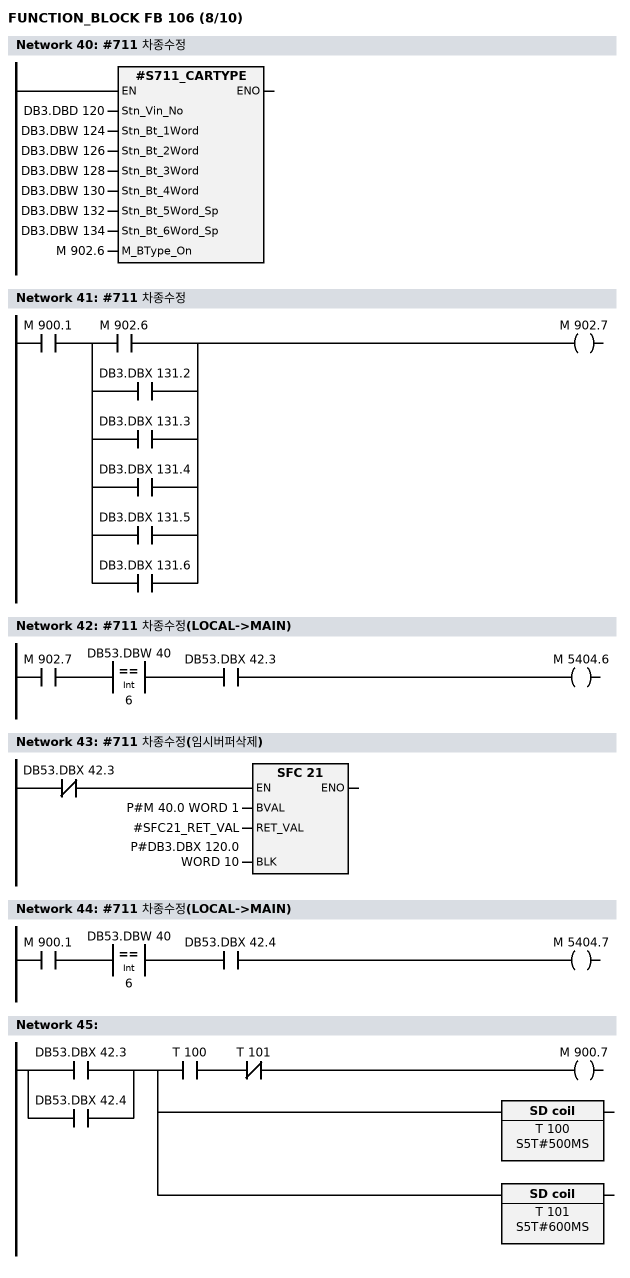

      CALL #S711_CARTYPE (
           Stn_Vin_No               := DB3.DBD  120,
           Stn_Bt_1Word             := DB3.DBW  124,
           Stn_Bt_2Word             := DB3.DBW  126,
           Stn_Bt_3Word             := DB3.DBW  128,
           Stn_Bt_4Word             := DB3.DBW  130,
           Stn_Bt_5Word_Sp          := DB3.DBW  132,
           Stn_Bt_6Word_Sp          := DB3.DBW  134,
           M_BType_On               := M    902.6);

      NOP   0;
NETWORK
TITLE =#711 차종수정

      A     M    900.1;
      A(    ;
      O     M    902.6;
      O     DB3.DBX  131.2;
      O     DB3.DBX  131.3;
      O     DB3.DBX  131.4;
      O     DB3.DBX  131.5;
      O     DB3.DBX  131.6;
      )     ;
      =     M    902.7;
NETWORK
TITLE =#711 차종수정(LOCAL->MAIN)

      A     M    902.7;
      A(    ;
      L     DB53.DBW   40;
      L     6;
      ==I   ;
      )     ;
      A     DB53.DBX   42.3;
      =     M   5404.6;
NETWORK
TITLE =#711 차종수정(임시버퍼삭제)

      AN    DB53.DBX   42.3;
      JNB   _00c;
      CALL SFC   21 (
           BVAL                     := P#M 40.0 WORD 1,
           RET_VAL                  := #SFC21_RET_VAL,
           BLK                      := P#DB3.DBX 120.0 WORD 10);
_00c: NOP   0;
NETWORK
TITLE =#711 차종수정(LOCAL->MAIN)

      A     M    900.1;
      A(    ;
      L     DB53.DBW   40;
      L     6;
      ==I   ;
      )     ;
      A     DB53.DBX   42.4;
      =     M   5404.7;
NETWORK
TITLE =

      O     DB53.DBX   42.3;
      O     DB53.DBX   42.4;
      =     L      2.0;
      A     L      2.0;
      A     T    100;
      AN    T    101;
      =     M    900.7;
      A     L      2.0;
      BLD   102;
      L     S5T#500MS;
      SD    T    100;
      A     L      2.0;
      BLD   102;
      L     S5T#600MS;
      SD    T    101;
NETWORK
TITLE =
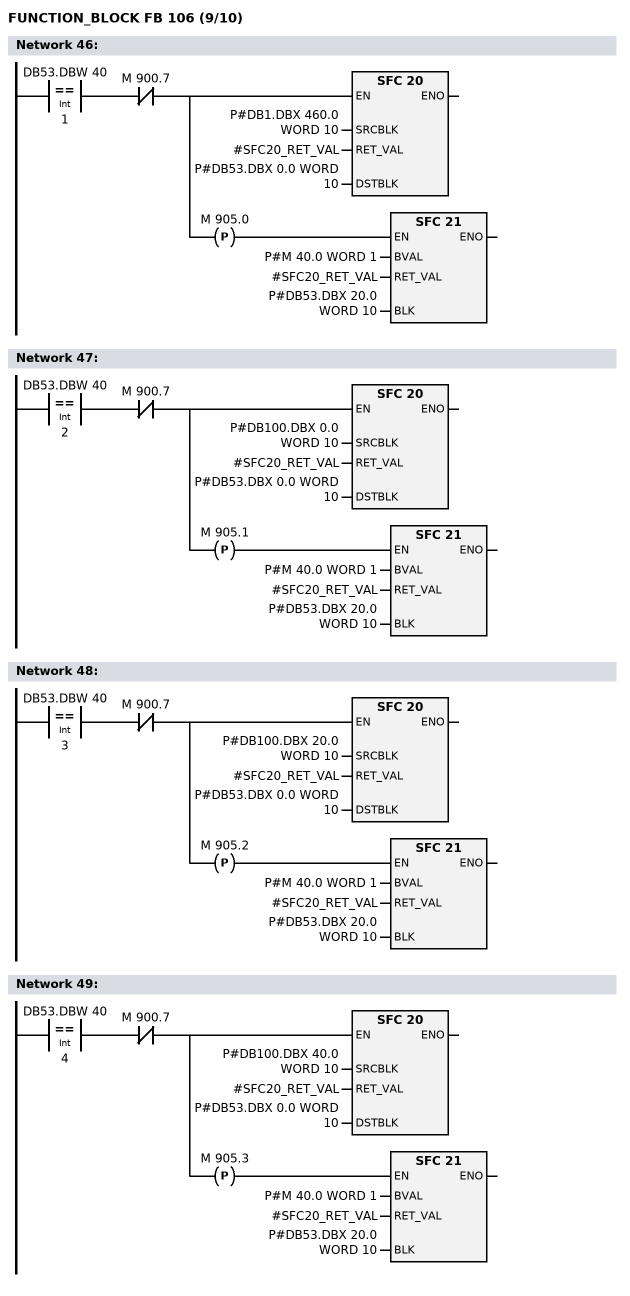

      A(    ;
      L     DB53.DBW   40;
      L     1;
      ==I   ;
      )     ;
      AN    M    900.7;
      =     L      2.0;
      A     L      2.0;
      JNB   _00d;
      CALL SFC   20 (
           SRCBLK                   := P#DB1.DBX 460.0 WORD 10,
           RET_VAL                  := #SFC20_RET_VAL,
           DSTBLK                   := P#DB53.DBX 0.0 WORD 10);
_00d: NOP   0;
      A     L      2.0;
      FP    M    905.0;
      JNB   _00e;
      CALL SFC   21 (
           BVAL                     := P#M 40.0 WORD 1,
           RET_VAL                  := #SFC20_RET_VAL,
           BLK                      := P#DB53.DBX 20.0 WORD 10);
_00e: NOP   0;
NETWORK
TITLE =

      A(    ;
      L     DB53.DBW   40;
      L     2;
      ==I   ;
      )     ;
      AN    M    900.7;
      =     L      2.0;
      A     L      2.0;
      JNB   _00f;
      CALL SFC   20 (
           SRCBLK                   := P#DB100.DBX 0.0 WORD 10,
           RET_VAL                  := #SFC20_RET_VAL,
           DSTBLK                   := P#DB53.DBX 0.0 WORD 10);
_00f: NOP   0;
      A     L      2.0;
      FP    M    905.1;
      JNB   _010;
      CALL SFC   21 (
           BVAL                     := P#M 40.0 WORD 1,
           RET_VAL                  := #SFC20_RET_VAL,
           BLK                      := P#DB53.DBX 20.0 WORD 10);
_010: NOP   0;
NETWORK
TITLE =

      A(    ;
      L     DB53.DBW   40;
      L     3;
      ==I   ;
      )     ;
      AN    M    900.7;
      =     L      2.0;
      A     L      2.0;
      JNB   _011;
      CALL SFC   20 (
           SRCBLK                   := P#DB100.DBX 20.0 WORD 10,
           RET_VAL                  := #SFC20_RET_VAL,
           DSTBLK                   := P#DB53.DBX 0.0 WORD 10);
_011: NOP   0;
      A     L      2.0;
      FP    M    905.2;
      JNB   _012;
      CALL SFC   21 (
           BVAL                     := P#M 40.0 WORD 1,
           RET_VAL                  := #SFC20_RET_VAL,
           BLK                      := P#DB53.DBX 20.0 WORD 10);
_012: NOP   0;
NETWORK
TITLE =

      A(    ;
      L     DB53.DBW   40;
      L     4;
      ==I   ;
      )     ;
      AN    M    900.7;
      =     L      2.0;
      A     L      2.0;
      JNB   _013;
      CALL SFC   20 (
           SRCBLK                   := P#DB100.DBX 40.0 WORD 10,
           RET_VAL                  := #SFC20_RET_VAL,
           DSTBLK                   := P#DB53.DBX 0.0 WORD 10);
_013: NOP   0;
      A     L      2.0;
      FP    M    905.3;
      JNB   _014;
      CALL SFC   21 (
           BVAL                     := P#M 40.0 WORD 1,
           RET_VAL                  := #SFC20_RET_VAL,
           BLK                      := P#DB53.DBX 20.0 WORD 10);
_014: NOP   0;
NETWORK
TITLE =
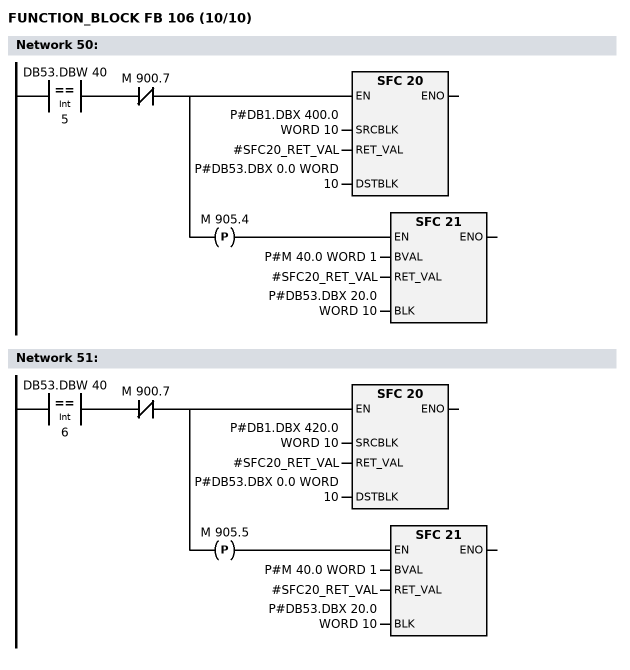

      A(    ;
      L     DB53.DBW   40;
      L     5;
      ==I   ;
      )     ;
      AN    M    900.7;
      =     L      2.0;
      A     L      2.0;
      JNB   _015;
      CALL SFC   20 (
           SRCBLK                   := P#DB1.DBX 400.0 WORD 10,
           RET_VAL                  := #SFC20_RET_VAL,
           DSTBLK                   := P#DB53.DBX 0.0 WORD 10);
_015: NOP   0;
      A     L      2.0;
      FP    M    905.4;
      JNB   _016;
      CALL SFC   21 (
           BVAL                     := P#M 40.0 WORD 1,
           RET_VAL                  := #SFC20_RET_VAL,
           BLK                      := P#DB53.DBX 20.0 WORD 10);
_016: NOP   0;
NETWORK
TITLE =

      A(    ;
      L     DB53.DBW   40;
      L     6;
      ==I   ;
      )     ;
      AN    M    900.7;
      =     L      2.0;
      A     L      2.0;
      JNB   _017;
      CALL SFC   20 (
           SRCBLK                   := P#DB1.DBX 420.0 WORD 10,
           RET_VAL                  := #SFC20_RET_VAL,
           DSTBLK                   := P#DB53.DBX 0.0 WORD 10);
_017: NOP   0;
      A     L      2.0;
      FP    M    905.5;
      JNB   _018;
      CALL SFC   21 (
           BVAL                     := P#M 40.0 WORD 1,
           RET_VAL                  := #SFC20_RET_VAL,
           BLK                      := P#DB53.DBX 20.0 WORD 10);
_018: NOP   0;
END_FUNCTION_BLOCK

DATA_BLOCK DB 106
TITLE =
VERSION : 0.0

 FB 106
BEGIN
   CAR_TYPE_MODIFY.Station := 0;
   CAR_TYPE_MODIFY.HMI_Disp_DB := 0;
   CAR_TYPE_MODIFY.HMI_Disp_Add := 0;
   CAR_TYPE_MODIFY.CType_DB := 0;
   CAR_TYPE_MODIFY.CType_Start_Add := 0;
   CAR_TYPE_MODIFY.Byte_per_Stn := 0;
   CAR_TYPE_MODIFY.M_Modify_OK := FALSE;
   CAR_TYPE_MODIFY.SS_CCR_On := FALSE;
   CAR_TYPE_MODIFY.PB_Set := FALSE;
   CAR_TYPE_MODIFY.PB_Reset := FALSE;
   CAR_TYPE_MODIFY.LP_CCR_On := FALSE;
   CAR_TYPE_MODIFY.LP_Modify_On := FALSE;
   CAR_TYPE_MODIFY.Source_Data := W#16#0;
   CAR_TYPE_MODIFY.Modify_Data := W#16#0;
   CAR_TYPE_MODIFY.Pre_Station := 0;
   CAR_TYPE_MODIFY.Station_PLS := FALSE;
   CAR_TYPE_MODIFY.Source_Add := 0;
   CAR_TYPE_MODIFY.SFC20_Ret := 0;
   CAR_TYPE_MODIFY.Fill_Source := W#16#0;
   SFC20_RET_VAL := 0;
   HMI_CAR_TYPE_V2.Stn_Vin_No := L#0;
   HMI_CAR_TYPE_V2.Stn_Bt_1Word := W#16#0;
   HMI_CAR_TYPE_V2.Stn_Bt_2Word := W#16#0;
   HMI_CAR_TYPE_V2.Stn_Bt_3Word := W#16#0;
   HMI_CAR_TYPE_V2.Stn_Bt_4Word := W#16#0;
   HMI_CAR_TYPE_V2.Stn_Bt_5Word_Sp := W#16#0;
   HMI_CAR_TYPE_V2.Stn_Bt_6Word_Sp := W#16#0;
   HMI_CAR_TYPE_V2.M_BType_On := FALSE;
   HMI_CAR_TYPE_V2.M_BType_None := FALSE;
   HMI_CAR_TYPE_V2.M_Bypass_BType := FALSE;
   HMI_CAR_TYPE_V2.M_BType_TL := FALSE;
   HMI_CAR_TYPE_V2.M_BType_LM := FALSE;
   HMI_CAR_TYPE_V2.M_BType_SP1 := FALSE;
   HMI_CAR_TYPE_V2.M_BType_SP2 := FALSE;
   HMI_CAR_TYPE_V2.M_BType_SP3 := FALSE;
   HMI_CAR_TYPE_V2.M_BType_DOM := FALSE;
   HMI_CAR_TYPE_V2.M_BType_EXP := FALSE;
   HMI_CAR_TYPE_V2.Robot_Prog_No := 0;
   HMI_CAR_TYPE_V2.STN_Btype_1Arr[0] := FALSE;
   HMI_CAR_TYPE_V2.STN_Btype_1Arr[1] := FALSE;
   HMI_CAR_TYPE_V2.STN_Btype_1Arr[2] := FALSE;
   HMI_CAR_TYPE_V2.STN_Btype_1Arr[3] := FALSE;
   HMI_CAR_TYPE_V2.STN_Btype_1Arr[4] := FALSE;
   HMI_CAR_TYPE_V2.STN_Btype_1Arr[5] := FALSE;
   HMI_CAR_TYPE_V2.STN_Btype_1Arr[6] := FALSE;
   HMI_CAR_TYPE_V2.STN_Btype_1Arr[7] := FALSE;
   HMI_CAR_TYPE_V2.STN_Btype_1Arr[8] := FALSE;
   HMI_CAR_TYPE_V2.STN_Btype_1Arr[9] := FALSE;
   HMI_CAR_TYPE_V2.STN_Btype_1Arr[10] := FALSE;
   HMI_CAR_TYPE_V2.STN_Btype_1Arr[11] := FALSE;
   HMI_CAR_TYPE_V2.STN_Btype_1Arr[12] := FALSE;
   HMI_CAR_TYPE_V2.STN_Btype_1Arr[13] := FALSE;
   HMI_CAR_TYPE_V2.STN_Btype_1Arr[14] := FALSE;
   HMI_CAR_TYPE_V2.STN_Btype_1Arr[15] := FALSE;
   HMI_CAR_TYPE_V2.STN_Btype_2Arr[0] := FALSE;
   HMI_CAR_TYPE_V2.STN_Btype_2Arr[1] := FALSE;
   HMI_CAR_TYPE_V2.STN_Btype_2Arr[2] := FALSE;
   HMI_CAR_TYPE_V2.STN_Btype_2Arr[3] := FALSE;
   HMI_CAR_TYPE_V2.STN_Btype_2Arr[4] := FALSE;
   HMI_CAR_TYPE_V2.STN_Btype_2Arr[5] := FALSE;
   HMI_CAR_TYPE_V2.STN_Btype_2Arr[6] := FALSE;
   HMI_CAR_TYPE_V2.STN_Btype_2Arr[7] := FALSE;
   HMI_CAR_TYPE_V2.STN_Btype_2Arr[8] := FALSE;
   HMI_CAR_TYPE_V2.STN_Btype_2Arr[9] := FALSE;
   HMI_CAR_TYPE_V2.STN_Btype_2Arr[10] := FALSE;
   HMI_CAR_TYPE_V2.STN_Btype_2Arr[11] := FALSE;
   HMI_CAR_TYPE_V2.STN_Btype_2Arr[12] := FALSE;
   HMI_CAR_TYPE_V2.STN_Btype_2Arr[13] := FALSE;
   HMI_CAR_TYPE_V2.STN_Btype_2Arr[14] := FALSE;
   HMI_CAR_TYPE_V2.STN_Btype_2Arr[15] := FALSE;
   HMI_CAR_TYPE_V2.STN_Btype_3Arr[0] := FALSE;
   HMI_CAR_TYPE_V2.STN_Btype_3Arr[1] := FALSE;
   HMI_CAR_TYPE_V2.STN_Btype_3Arr[2] := FALSE;
   HMI_CAR_TYPE_V2.STN_Btype_3Arr[3] := FALSE;
   HMI_CAR_TYPE_V2.STN_Btype_3Arr[4] := FALSE;
   HMI_CAR_TYPE_V2.STN_Btype_3Arr[5] := FALSE;
   HMI_CAR_TYPE_V2.STN_Btype_3Arr[6] := FALSE;
   HMI_CAR_TYPE_V2.STN_Btype_3Arr[7] := FALSE;
   HMI_CAR_TYPE_V2.STN_Btype_3Arr[8] := FALSE;
   HMI_CAR_TYPE_V2.STN_Btype_3Arr[9] := FALSE;
   HMI_CAR_TYPE_V2.STN_Btype_3Arr[10] := FALSE;
   HMI_CAR_TYPE_V2.STN_Btype_3Arr[11] := FALSE;
   HMI_CAR_TYPE_V2.STN_Btype_3Arr[12] := FALSE;
   HMI_CAR_TYPE_V2.STN_Btype_3Arr[13] := FALSE;
   HMI_CAR_TYPE_V2.STN_Btype_3Arr[14] := FALSE;
   HMI_CAR_TYPE_V2.STN_Btype_3Arr[15] := FALSE;
   HMI_CAR_TYPE_V2.STN_Btype_4Arr[0] := FALSE;
   HMI_CAR_TYPE_V2.STN_Btype_4Arr[1] := FALSE;
   HMI_CAR_TYPE_V2.STN_Btype_4Arr[2] := FALSE;
   HMI_CAR_TYPE_V2.STN_Btype_4Arr[3] := FALSE;
   HMI_CAR_TYPE_V2.STN_Btype_4Arr[4] := FALSE;
   HMI_CAR_TYPE_V2.STN_Btype_4Arr[5] := FALSE;
   HMI_CAR_TYPE_V2.STN_Btype_4Arr[6] := FALSE;
   HMI_CAR_TYPE_V2.STN_Btype_4Arr[7] := FALSE;
   HMI_CAR_TYPE_V2.STN_Btype_4Arr[8] := FALSE;
   HMI_CAR_TYPE_V2.STN_Btype_4Arr[9] := FALSE;
   HMI_CAR_TYPE_V2.STN_Btype_4Arr[10] := FALSE;
   HMI_CAR_TYPE_V2.STN_Btype_4Arr[11] := FALSE;
   HMI_CAR_TYPE_V2.STN_Btype_4Arr[12] := FALSE;
   HMI_CAR_TYPE_V2.STN_Btype_4Arr[13] := FALSE;
   HMI_CAR_TYPE_V2.STN_Btype_4Arr[14] := FALSE;
   HMI_CAR_TYPE_V2.STN_Btype_4Arr[15] := FALSE;
   HMI_CAR_TYPE_V2.STN_Btype_5Arr[0] := FALSE;
   HMI_CAR_TYPE_V2.STN_Btype_5Arr[1] := FALSE;
   HMI_CAR_TYPE_V2.STN_Btype_5Arr[2] := FALSE;
   HMI_CAR_TYPE_V2.STN_Btype_5Arr[3] := FALSE;
   HMI_CAR_TYPE_V2.STN_Btype_5Arr[4] := FALSE;
   HMI_CAR_TYPE_V2.STN_Btype_5Arr[5] := FALSE;
   HMI_CAR_TYPE_V2.STN_Btype_5Arr[6] := FALSE;
   HMI_CAR_TYPE_V2.STN_Btype_5Arr[7] := FALSE;
   HMI_CAR_TYPE_V2.STN_Btype_5Arr[8] := FALSE;
   HMI_CAR_TYPE_V2.STN_Btype_5Arr[9] := FALSE;
   HMI_CAR_TYPE_V2.STN_Btype_5Arr[10] := FALSE;
   HMI_CAR_TYPE_V2.STN_Btype_5Arr[11] := FALSE;
   HMI_CAR_TYPE_V2.STN_Btype_5Arr[12] := FALSE;
   HMI_CAR_TYPE_V2.STN_Btype_5Arr[13] := FALSE;
   HMI_CAR_TYPE_V2.STN_Btype_5Arr[14] := FALSE;
   HMI_CAR_TYPE_V2.STN_Btype_5Arr[15] := FALSE;
   HMI_CAR_TYPE_V2.STN_Btype_6Arr[0] := FALSE;
   HMI_CAR_TYPE_V2.STN_Btype_6Arr[1] := FALSE;
   HMI_CAR_TYPE_V2.STN_Btype_6Arr[2] := FALSE;
   HMI_CAR_TYPE_V2.STN_Btype_6Arr[3] := FALSE;
   HMI_CAR_TYPE_V2.STN_Btype_6Arr[4] := FALSE;
   HMI_CAR_TYPE_V2.STN_Btype_6Arr[5] := FALSE;
   HMI_CAR_TYPE_V2.STN_Btype_6Arr[6] := FALSE;
   HMI_CAR_TYPE_V2.STN_Btype_6Arr[7] := FALSE;
   HMI_CAR_TYPE_V2.STN_Btype_6Arr[8] := FALSE;
   HMI_CAR_TYPE_V2.STN_Btype_6Arr[9] := FALSE;
   HMI_CAR_TYPE_V2.STN_Btype_6Arr[10] := FALSE;
   HMI_CAR_TYPE_V2.STN_Btype_6Arr[11] := FALSE;
   HMI_CAR_TYPE_V2.STN_Btype_6Arr[12] := FALSE;
   HMI_CAR_TYPE_V2.STN_Btype_6Arr[13] := FALSE;
   HMI_CAR_TYPE_V2.STN_Btype_6Arr[14] := FALSE;
   HMI_CAR_TYPE_V2.STN_Btype_6Arr[15] := FALSE;
   HMI_CAR_TYPE_V2.STN_1st_BT_On := FALSE;
   HMI_CAR_TYPE_V2.STN_2nd_BT_On := FALSE;
   HMI_CAR_TYPE_V2.STN_3rd_BT_On := FALSE;
   HMI_CAR_TYPE_V2.STN_4th_BT_On := FALSE;
   HMI_CAR_TYPE_V2.STN_5th_BT_On := FALSE;
   HMI_CAR_TYPE_V2.STN_6th_BT_On := FALSE;
   HMI_CAR_TYPE_V2.STN_7th_BT_On := FALSE;
   HMI_CAR_TYPE_V2.STN_8th_BT_On := FALSE;
   HMI_CAR_TYPE_V2.STN_9th_BT_On := FALSE;
   HMI_CAR_TYPE_V2.STN_10th_BT_On := FALSE;
   HMI_CAR_TYPE_V2.STN_11th_BT_On := FALSE;
   HMI_CAR_TYPE_V2.STN_12th_BT_On := FALSE;
   HMI_CAR_TYPE_V2.STN_1st_BT_Off := FALSE;
   HMI_CAR_TYPE_V2.BLKMove_Ret := 0;
   HMI_CAR_TYPE_V2.VIN_1BCD := W#16#0;
   HMI_CAR_TYPE_V2.VIN_2BCD := W#16#0;
   HMI_CAR_TYPE_V2.VIN_1Int := 0;
   HMI_CAR_TYPE_V2.VIN_2Int := 0;
   S6_HMI_CAR_TYPE_V2.Stn_Vin_No := L#0;
   S6_HMI_CAR_TYPE_V2.Stn_Bt_1Word := W#16#0;
   S6_HMI_CAR_TYPE_V2.Stn_Bt_2Word := W#16#0;
   S6_HMI_CAR_TYPE_V2.Stn_Bt_3Word := W#16#0;
   S6_HMI_CAR_TYPE_V2.Stn_Bt_4Word := W#16#0;
   S6_HMI_CAR_TYPE_V2.Stn_Bt_5Word_Sp := W#16#0;
   S6_HMI_CAR_TYPE_V2.Stn_Bt_6Word_Sp := W#16#0;
   S6_HMI_CAR_TYPE_V2.M_BType_On := FALSE;
   S6_HMI_CAR_TYPE_V2.M_BType_None := FALSE;
   S6_HMI_CAR_TYPE_V2.M_Bypass_BType := FALSE;
   S6_HMI_CAR_TYPE_V2.M_BType_TL := FALSE;
   S6_HMI_CAR_TYPE_V2.M_BType_LM := FALSE;
   S6_HMI_CAR_TYPE_V2.M_BType_SP1 := FALSE;
   S6_HMI_CAR_TYPE_V2.M_BType_SP2 := FALSE;
   S6_HMI_CAR_TYPE_V2.M_BType_SP3 := FALSE;
   S6_HMI_CAR_TYPE_V2.M_BType_DOM := FALSE;
   S6_HMI_CAR_TYPE_V2.M_BType_EXP := FALSE;
   S6_HMI_CAR_TYPE_V2.Robot_Prog_No := 0;
   S6_HMI_CAR_TYPE_V2.STN_Btype_1Arr[0] := FALSE;
   S6_HMI_CAR_TYPE_V2.STN_Btype_1Arr[1] := FALSE;
   S6_HMI_CAR_TYPE_V2.STN_Btype_1Arr[2] := FALSE;
   S6_HMI_CAR_TYPE_V2.STN_Btype_1Arr[3] := FALSE;
   S6_HMI_CAR_TYPE_V2.STN_Btype_1Arr[4] := FALSE;
   S6_HMI_CAR_TYPE_V2.STN_Btype_1Arr[5] := FALSE;
   S6_HMI_CAR_TYPE_V2.STN_Btype_1Arr[6] := FALSE;
   S6_HMI_CAR_TYPE_V2.STN_Btype_1Arr[7] := FALSE;
   S6_HMI_CAR_TYPE_V2.STN_Btype_1Arr[8] := FALSE;
   S6_HMI_CAR_TYPE_V2.STN_Btype_1Arr[9] := FALSE;
   S6_HMI_CAR_TYPE_V2.STN_Btype_1Arr[10] := FALSE;
   S6_HMI_CAR_TYPE_V2.STN_Btype_1Arr[11] := FALSE;
   S6_HMI_CAR_TYPE_V2.STN_Btype_1Arr[12] := FALSE;
   S6_HMI_CAR_TYPE_V2.STN_Btype_1Arr[13] := FALSE;
   S6_HMI_CAR_TYPE_V2.STN_Btype_1Arr[14] := FALSE;
   S6_HMI_CAR_TYPE_V2.STN_Btype_1Arr[15] := FALSE;
   S6_HMI_CAR_TYPE_V2.STN_Btype_2Arr[0] := FALSE;
   S6_HMI_CAR_TYPE_V2.STN_Btype_2Arr[1] := FALSE;
   S6_HMI_CAR_TYPE_V2.STN_Btype_2Arr[2] := FALSE;
   S6_HMI_CAR_TYPE_V2.STN_Btype_2Arr[3] := FALSE;
   S6_HMI_CAR_TYPE_V2.STN_Btype_2Arr[4] := FALSE;
   S6_HMI_CAR_TYPE_V2.STN_Btype_2Arr[5] := FALSE;
   S6_HMI_CAR_TYPE_V2.STN_Btype_2Arr[6] := FALSE;
   S6_HMI_CAR_TYPE_V2.STN_Btype_2Arr[7] := FALSE;
   S6_HMI_CAR_TYPE_V2.STN_Btype_2Arr[8] := FALSE;
   S6_HMI_CAR_TYPE_V2.STN_Btype_2Arr[9] := FALSE;
   S6_HMI_CAR_TYPE_V2.STN_Btype_2Arr[10] := FALSE;
   S6_HMI_CAR_TYPE_V2.STN_Btype_2Arr[11] := FALSE;
   S6_HMI_CAR_TYPE_V2.STN_Btype_2Arr[12] := FALSE;
   S6_HMI_CAR_TYPE_V2.STN_Btype_2Arr[13] := FALSE;
   S6_HMI_CAR_TYPE_V2.STN_Btype_2Arr[14] := FALSE;
   S6_HMI_CAR_TYPE_V2.STN_Btype_2Arr[15] := FALSE;
   S6_HMI_CAR_TYPE_V2.STN_Btype_3Arr[0] := FALSE;
   S6_HMI_CAR_TYPE_V2.STN_Btype_3Arr[1] := FALSE;
   S6_HMI_CAR_TYPE_V2.STN_Btype_3Arr[2] := FALSE;
   S6_HMI_CAR_TYPE_V2.STN_Btype_3Arr[3] := FALSE;
   S6_HMI_CAR_TYPE_V2.STN_Btype_3Arr[4] := FALSE;
   S6_HMI_CAR_TYPE_V2.STN_Btype_3Arr[5] := FALSE;
   S6_HMI_CAR_TYPE_V2.STN_Btype_3Arr[6] := FALSE;
   S6_HMI_CAR_TYPE_V2.STN_Btype_3Arr[7] := FALSE;
   S6_HMI_CAR_TYPE_V2.STN_Btype_3Arr[8] := FALSE;
   S6_HMI_CAR_TYPE_V2.STN_Btype_3Arr[9] := FALSE;
   S6_HMI_CAR_TYPE_V2.STN_Btype_3Arr[10] := FALSE;
   S6_HMI_CAR_TYPE_V2.STN_Btype_3Arr[11] := FALSE;
   S6_HMI_CAR_TYPE_V2.STN_Btype_3Arr[12] := FALSE;
   S6_HMI_CAR_TYPE_V2.STN_Btype_3Arr[13] := FALSE;
   S6_HMI_CAR_TYPE_V2.STN_Btype_3Arr[14] := FALSE;
   S6_HMI_CAR_TYPE_V2.STN_Btype_3Arr[15] := FALSE;
   S6_HMI_CAR_TYPE_V2.STN_Btype_4Arr[0] := FALSE;
   S6_HMI_CAR_TYPE_V2.STN_Btype_4Arr[1] := FALSE;
   S6_HMI_CAR_TYPE_V2.STN_Btype_4Arr[2] := FALSE;
   S6_HMI_CAR_TYPE_V2.STN_Btype_4Arr[3] := FALSE;
   S6_HMI_CAR_TYPE_V2.STN_Btype_4Arr[4] := FALSE;
   S6_HMI_CAR_TYPE_V2.STN_Btype_4Arr[5] := FALSE;
   S6_HMI_CAR_TYPE_V2.STN_Btype_4Arr[6] := FALSE;
   S6_HMI_CAR_TYPE_V2.STN_Btype_4Arr[7] := FALSE;
   S6_HMI_CAR_TYPE_V2.STN_Btype_4Arr[8] := FALSE;
   S6_HMI_CAR_TYPE_V2.STN_Btype_4Arr[9] := FALSE;
   S6_HMI_CAR_TYPE_V2.STN_Btype_4Arr[10] := FALSE;
   S6_HMI_CAR_TYPE_V2.STN_Btype_4Arr[11] := FALSE;
   S6_HMI_CAR_TYPE_V2.STN_Btype_4Arr[12] := FALSE;
   S6_HMI_CAR_TYPE_V2.STN_Btype_4Arr[13] := FALSE;
   S6_HMI_CAR_TYPE_V2.STN_Btype_4Arr[14] := FALSE;
   S6_HMI_CAR_TYPE_V2.STN_Btype_4Arr[15] := FALSE;
   S6_HMI_CAR_TYPE_V2.STN_Btype_5Arr[0] := FALSE;
   S6_HMI_CAR_TYPE_V2.STN_Btype_5Arr[1] := FALSE;
   S6_HMI_CAR_TYPE_V2.STN_Btype_5Arr[2] := FALSE;
   S6_HMI_CAR_TYPE_V2.STN_Btype_5Arr[3] := FALSE;
   S6_HMI_CAR_TYPE_V2.STN_Btype_5Arr[4] := FALSE;
   S6_HMI_CAR_TYPE_V2.STN_Btype_5Arr[5] := FALSE;
   S6_HMI_CAR_TYPE_V2.STN_Btype_5Arr[6] := FALSE;
   S6_HMI_CAR_TYPE_V2.STN_Btype_5Arr[7] := FALSE;
   S6_HMI_CAR_TYPE_V2.STN_Btype_5Arr[8] := FALSE;
   S6_HMI_CAR_TYPE_V2.STN_Btype_5Arr[9] := FALSE;
   S6_HMI_CAR_TYPE_V2.STN_Btype_5Arr[10] := FALSE;
   S6_HMI_CAR_TYPE_V2.STN_Btype_5Arr[11] := FALSE;
   S6_HMI_CAR_TYPE_V2.STN_Btype_5Arr[12] := FALSE;
   S6_HMI_CAR_TYPE_V2.STN_Btype_5Arr[13] := FALSE;
   S6_HMI_CAR_TYPE_V2.STN_Btype_5Arr[14] := FALSE;
   S6_HMI_CAR_TYPE_V2.STN_Btype_5Arr[15] := FALSE;
   S6_HMI_CAR_TYPE_V2.STN_Btype_6Arr[0] := FALSE;
   S6_HMI_CAR_TYPE_V2.STN_Btype_6Arr[1] := FALSE;
   S6_HMI_CAR_TYPE_V2.STN_Btype_6Arr[2] := FALSE;
   S6_HMI_CAR_TYPE_V2.STN_Btype_6Arr[3] := FALSE;
   S6_HMI_CAR_TYPE_V2.STN_Btype_6Arr[4] := FALSE;
   S6_HMI_CAR_TYPE_V2.STN_Btype_6Arr[5] := FALSE;
   S6_HMI_CAR_TYPE_V2.STN_Btype_6Arr[6] := FALSE;
   S6_HMI_CAR_TYPE_V2.STN_Btype_6Arr[7] := FALSE;
   S6_HMI_CAR_TYPE_V2.STN_Btype_6Arr[8] := FALSE;
   S6_HMI_CAR_TYPE_V2.STN_Btype_6Arr[9] := FALSE;
   S6_HMI_CAR_TYPE_V2.STN_Btype_6Arr[10] := FALSE;
   S6_HMI_CAR_TYPE_V2.STN_Btype_6Arr[11] := FALSE;
   S6_HMI_CAR_TYPE_V2.STN_Btype_6Arr[12] := FALSE;
   S6_HMI_CAR_TYPE_V2.STN_Btype_6Arr[13] := FALSE;
   S6_HMI_CAR_TYPE_V2.STN_Btype_6Arr[14] := FALSE;
   S6_HMI_CAR_TYPE_V2.STN_Btype_6Arr[15] := FALSE;
   S6_HMI_CAR_TYPE_V2.STN_1st_BT_On := FALSE;
   S6_HMI_CAR_TYPE_V2.STN_2nd_BT_On := FALSE;
   S6_HMI_CAR_TYPE_V2.STN_3rd_BT_On := FALSE;
   S6_HMI_CAR_TYPE_V2.STN_4th_BT_On := FALSE;
   S6_HMI_CAR_TYPE_V2.STN_5th_BT_On := FALSE;
   S6_HMI_CAR_TYPE_V2.STN_6th_BT_On := FALSE;
   S6_HMI_CAR_TYPE_V2.STN_7th_BT_On := FALSE;
   S6_HMI_CAR_TYPE_V2.STN_8th_BT_On := FALSE;
   S6_HMI_CAR_TYPE_V2.STN_9th_BT_On := FALSE;
   S6_HMI_CAR_TYPE_V2.STN_10th_BT_On := FALSE;
   S6_HMI_CAR_TYPE_V2.STN_11th_BT_On := FALSE;
   S6_HMI_CAR_TYPE_V2.STN_12th_BT_On := FALSE;
   S6_HMI_CAR_TYPE_V2.STN_1st_BT_Off := FALSE;
   S6_HMI_CAR_TYPE_V2.BLKMove_Ret := 0;
   S6_HMI_CAR_TYPE_V2.VIN_1BCD := W#16#0;
   S6_HMI_CAR_TYPE_V2.VIN_2BCD := W#16#0;
   S6_HMI_CAR_TYPE_V2.VIN_1Int := 0;
   S6_HMI_CAR_TYPE_V2.VIN_2Int := 0;
   S6_CAR_TYPE_MODIFY.Station := 0;
   S6_CAR_TYPE_MODIFY.HMI_Disp_DB := 0;
   S6_CAR_TYPE_MODIFY.HMI_Disp_Add := 0;
   S6_CAR_TYPE_MODIFY.CType_DB := 0;
   S6_CAR_TYPE_MODIFY.CType_Start_Add := 0;
   S6_CAR_TYPE_MODIFY.Byte_per_Stn := 0;
   S6_CAR_TYPE_MODIFY.M_Modify_OK := FALSE;
   S6_CAR_TYPE_MODIFY.SS_CCR_On := FALSE;
   S6_CAR_TYPE_MODIFY.PB_Set := FALSE;
   S6_CAR_TYPE_MODIFY.PB_Reset := FALSE;
   S6_CAR_TYPE_MODIFY.LP_CCR_On := FALSE;
   S6_CAR_TYPE_MODIFY.LP_Modify_On := FALSE;
   S6_CAR_TYPE_MODIFY.Source_Data := W#16#0;
   S6_CAR_TYPE_MODIFY.Modify_Data := W#16#0;
   S6_CAR_TYPE_MODIFY.Pre_Station := 0;
   S6_CAR_TYPE_MODIFY.Station_PLS := FALSE;
   S6_CAR_TYPE_MODIFY.Source_Add := 0;
   S6_CAR_TYPE_MODIFY.SFC20_Ret := 0;
   S6_CAR_TYPE_MODIFY.Fill_Source := W#16#0;
   S486RH_CARTYPE.Stn_Vin_No := L#0;
   S486RH_CARTYPE.Stn_Bt_1Word := W#16#0;
   S486RH_CARTYPE.Stn_Bt_2Word := W#16#0;
   S486RH_CARTYPE.Stn_Bt_3Word := W#16#0;
   S486RH_CARTYPE.Stn_Bt_4Word := W#16#0;
   S486RH_CARTYPE.Stn_Bt_5Word_Sp := W#16#0;
   S486RH_CARTYPE.Stn_Bt_6Word_Sp := W#16#0;
   S486RH_CARTYPE.M_BType_On := FALSE;
   S486RH_CARTYPE.M_BType_None := FALSE;
   S486RH_CARTYPE.M_Bypass_BType := FALSE;
   S486RH_CARTYPE.M_BType_TL := FALSE;
   S486RH_CARTYPE.M_BType_LM := FALSE;
   S486RH_CARTYPE.M_BType_SP1 := FALSE;
   S486RH_CARTYPE.M_BType_SP2 := FALSE;
   S486RH_CARTYPE.M_BType_SP3 := FALSE;
   S486RH_CARTYPE.M_BType_DOM := FALSE;
   S486RH_CARTYPE.M_BType_EXP := FALSE;
   S486RH_CARTYPE.Robot_Prog_No := 0;
   S486RH_CARTYPE.STN_Btype_1Arr[0] := FALSE;
   S486RH_CARTYPE.STN_Btype_1Arr[1] := FALSE;
   S486RH_CARTYPE.STN_Btype_1Arr[2] := FALSE;
   S486RH_CARTYPE.STN_Btype_1Arr[3] := FALSE;
   S486RH_CARTYPE.STN_Btype_1Arr[4] := FALSE;
   S486RH_CARTYPE.STN_Btype_1Arr[5] := FALSE;
   S486RH_CARTYPE.STN_Btype_1Arr[6] := FALSE;
   S486RH_CARTYPE.STN_Btype_1Arr[7] := FALSE;
   S486RH_CARTYPE.STN_Btype_1Arr[8] := FALSE;
   S486RH_CARTYPE.STN_Btype_1Arr[9] := FALSE;
   S486RH_CARTYPE.STN_Btype_1Arr[10] := FALSE;
   S486RH_CARTYPE.STN_Btype_1Arr[11] := FALSE;
   S486RH_CARTYPE.STN_Btype_1Arr[12] := FALSE;
   S486RH_CARTYPE.STN_Btype_1Arr[13] := FALSE;
   S486RH_CARTYPE.STN_Btype_1Arr[14] := FALSE;
   S486RH_CARTYPE.STN_Btype_1Arr[15] := FALSE;
   S486RH_CARTYPE.STN_Btype_2Arr[0] := FALSE;
   S486RH_CARTYPE.STN_Btype_2Arr[1] := FALSE;
   S486RH_CARTYPE.STN_Btype_2Arr[2] := FALSE;
   S486RH_CARTYPE.STN_Btype_2Arr[3] := FALSE;
   S486RH_CARTYPE.STN_Btype_2Arr[4] := FALSE;
   S486RH_CARTYPE.STN_Btype_2Arr[5] := FALSE;
   S486RH_CARTYPE.STN_Btype_2Arr[6] := FALSE;
   S486RH_CARTYPE.STN_Btype_2Arr[7] := FALSE;
   S486RH_CARTYPE.STN_Btype_2Arr[8] := FALSE;
   S486RH_CARTYPE.STN_Btype_2Arr[9] := FALSE;
   S486RH_CARTYPE.STN_Btype_2Arr[10] := FALSE;
   S486RH_CARTYPE.STN_Btype_2Arr[11] := FALSE;
   S486RH_CARTYPE.STN_Btype_2Arr[12] := FALSE;
   S486RH_CARTYPE.STN_Btype_2Arr[13] := FALSE;
   S486RH_CARTYPE.STN_Btype_2Arr[14] := FALSE;
   S486RH_CARTYPE.STN_Btype_2Arr[15] := FALSE;
   S486RH_CARTYPE.STN_Btype_3Arr[0] := FALSE;
   S486RH_CARTYPE.STN_Btype_3Arr[1] := FALSE;
   S486RH_CARTYPE.STN_Btype_3Arr[2] := FALSE;
   S486RH_CARTYPE.STN_Btype_3Arr[3] := FALSE;
   S486RH_CARTYPE.STN_Btype_3Arr[4] := FALSE;
   S486RH_CARTYPE.STN_Btype_3Arr[5] := FALSE;
   S486RH_CARTYPE.STN_Btype_3Arr[6] := FALSE;
   S486RH_CARTYPE.STN_Btype_3Arr[7] := FALSE;
   S486RH_CARTYPE.STN_Btype_3Arr[8] := FALSE;
   S486RH_CARTYPE.STN_Btype_3Arr[9] := FALSE;
   S486RH_CARTYPE.STN_Btype_3Arr[10] := FALSE;
   S486RH_CARTYPE.STN_Btype_3Arr[11] := FALSE;
   S486RH_CARTYPE.STN_Btype_3Arr[12] := FALSE;
   S486RH_CARTYPE.STN_Btype_3Arr[13] := FALSE;
   S486RH_CARTYPE.STN_Btype_3Arr[14] := FALSE;
   S486RH_CARTYPE.STN_Btype_3Arr[15] := FALSE;
   S486RH_CARTYPE.STN_Btype_4Arr[0] := FALSE;
   S486RH_CARTYPE.STN_Btype_4Arr[1] := FALSE;
   S486RH_CARTYPE.STN_Btype_4Arr[2] := FALSE;
   S486RH_CARTYPE.STN_Btype_4Arr[3] := FALSE;
   S486RH_CARTYPE.STN_Btype_4Arr[4] := FALSE;
   S486RH_CARTYPE.STN_Btype_4Arr[5] := FALSE;
   S486RH_CARTYPE.STN_Btype_4Arr[6] := FALSE;
   S486RH_CARTYPE.STN_Btype_4Arr[7] := FALSE;
   S486RH_CARTYPE.STN_Btype_4Arr[8] := FALSE;
   S486RH_CARTYPE.STN_Btype_4Arr[9] := FALSE;
   S486RH_CARTYPE.STN_Btype_4Arr[10] := FALSE;
   S486RH_CARTYPE.STN_Btype_4Arr[11] := FALSE;
   S486RH_CARTYPE.STN_Btype_4Arr[12] := FALSE;
   S486RH_CARTYPE.STN_Btype_4Arr[13] := FALSE;
   S486RH_CARTYPE.STN_Btype_4Arr[14] := FALSE;
   S486RH_CARTYPE.STN_Btype_4Arr[15] := FALSE;
   S486RH_CARTYPE.STN_Btype_5Arr[0] := FALSE;
   S486RH_CARTYPE.STN_Btype_5Arr[1] := FALSE;
   S486RH_CARTYPE.STN_Btype_5Arr[2] := FALSE;
   S486RH_CARTYPE.STN_Btype_5Arr[3] := FALSE;
   S486RH_CARTYPE.STN_Btype_5Arr[4] := FALSE;
   S486RH_CARTYPE.STN_Btype_5Arr[5] := FALSE;
   S486RH_CARTYPE.STN_Btype_5Arr[6] := FALSE;
   S486RH_CARTYPE.STN_Btype_5Arr[7] := FALSE;
   S486RH_CARTYPE.STN_Btype_5Arr[8] := FALSE;
   S486RH_CARTYPE.STN_Btype_5Arr[9] := FALSE;
   S486RH_CARTYPE.STN_Btype_5Arr[10] := FALSE;
   S486RH_CARTYPE.STN_Btype_5Arr[11] := FALSE;
   S486RH_CARTYPE.STN_Btype_5Arr[12] := FALSE;
   S486RH_CARTYPE.STN_Btype_5Arr[13] := FALSE;
   S486RH_CARTYPE.STN_Btype_5Arr[14] := FALSE;
   S486RH_CARTYPE.STN_Btype_5Arr[15] := FALSE;
   S486RH_CARTYPE.STN_Btype_6Arr[0] := FALSE;
   S486RH_CARTYPE.STN_Btype_6Arr[1] := FALSE;
   S486RH_CARTYPE.STN_Btype_6Arr[2] := FALSE;
   S486RH_CARTYPE.STN_Btype_6Arr[3] := FALSE;
   S486RH_CARTYPE.STN_Btype_6Arr[4] := FALSE;
   S486RH_CARTYPE.STN_Btype_6Arr[5] := FALSE;
   S486RH_CARTYPE.STN_Btype_6Arr[6] := FALSE;
   S486RH_CARTYPE.STN_Btype_6Arr[7] := FALSE;
   S486RH_CARTYPE.STN_Btype_6Arr[8] := FALSE;
   S486RH_CARTYPE.STN_Btype_6Arr[9] := FALSE;
   S486RH_CARTYPE.STN_Btype_6Arr[10] := FALSE;
   S486RH_CARTYPE.STN_Btype_6Arr[11] := FALSE;
   S486RH_CARTYPE.STN_Btype_6Arr[12] := FALSE;
   S486RH_CARTYPE.STN_Btype_6Arr[13] := FALSE;
   S486RH_CARTYPE.STN_Btype_6Arr[14] := FALSE;
   S486RH_CARTYPE.STN_Btype_6Arr[15] := FALSE;
   S486RH_CARTYPE.STN_1st_BT_On := FALSE;
   S486RH_CARTYPE.STN_2nd_BT_On := FALSE;
   S486RH_CARTYPE.STN_3rd_BT_On := FALSE;
   S486RH_CARTYPE.STN_4th_BT_On := FALSE;
   S486RH_CARTYPE.STN_5th_BT_On := FALSE;
   S486RH_CARTYPE.STN_6th_BT_On := FALSE;
   S486RH_CARTYPE.STN_7th_BT_On := FALSE;
   S486RH_CARTYPE.STN_8th_BT_On := FALSE;
   S486RH_CARTYPE.STN_9th_BT_On := FALSE;
   S486RH_CARTYPE.STN_10th_BT_On := FALSE;
   S486RH_CARTYPE.STN_11th_BT_On := FALSE;
   S486RH_CARTYPE.STN_12th_BT_On := FALSE;
   S486RH_CARTYPE.STN_1st_BT_Off := FALSE;
   S486RH_CARTYPE.BLKMove_Ret := 0;
   S486RH_CARTYPE.VIN_1BCD := W#16#0;
   S486RH_CARTYPE.VIN_2BCD := W#16#0;
   S486RH_CARTYPE.VIN_1Int := 0;
   S486RH_CARTYPE.VIN_2Int := 0;
   S486LH_CARTYPE.Stn_Vin_No := L#0;
   S486LH_CARTYPE.Stn_Bt_1Word := W#16#0;
   S486LH_CARTYPE.Stn_Bt_2Word := W#16#0;
   S486LH_CARTYPE.Stn_Bt_3Word := W#16#0;
   S486LH_CARTYPE.Stn_Bt_4Word := W#16#0;
   S486LH_CARTYPE.Stn_Bt_5Word_Sp := W#16#0;
   S486LH_CARTYPE.Stn_Bt_6Word_Sp := W#16#0;
   S486LH_CARTYPE.M_BType_On := FALSE;
   S486LH_CARTYPE.M_BType_None := FALSE;
   S486LH_CARTYPE.M_Bypass_BType := FALSE;
   S486LH_CARTYPE.M_BType_TL := FALSE;
   S486LH_CARTYPE.M_BType_LM := FALSE;
   S486LH_CARTYPE.M_BType_SP1 := FALSE;
   S486LH_CARTYPE.M_BType_SP2 := FALSE;
   S486LH_CARTYPE.M_BType_SP3 := FALSE;
   S486LH_CARTYPE.M_BType_DOM := FALSE;
   S486LH_CARTYPE.M_BType_EXP := FALSE;
   S486LH_CARTYPE.Robot_Prog_No := 0;
   S486LH_CARTYPE.STN_Btype_1Arr[0] := FALSE;
   S486LH_CARTYPE.STN_Btype_1Arr[1] := FALSE;
   S486LH_CARTYPE.STN_Btype_1Arr[2] := FALSE;
   S486LH_CARTYPE.STN_Btype_1Arr[3] := FALSE;
   S486LH_CARTYPE.STN_Btype_1Arr[4] := FALSE;
   S486LH_CARTYPE.STN_Btype_1Arr[5] := FALSE;
   S486LH_CARTYPE.STN_Btype_1Arr[6] := FALSE;
   S486LH_CARTYPE.STN_Btype_1Arr[7] := FALSE;
   S486LH_CARTYPE.STN_Btype_1Arr[8] := FALSE;
   S486LH_CARTYPE.STN_Btype_1Arr[9] := FALSE;
   S486LH_CARTYPE.STN_Btype_1Arr[10] := FALSE;
   S486LH_CARTYPE.STN_Btype_1Arr[11] := FALSE;
   S486LH_CARTYPE.STN_Btype_1Arr[12] := FALSE;
   S486LH_CARTYPE.STN_Btype_1Arr[13] := FALSE;
   S486LH_CARTYPE.STN_Btype_1Arr[14] := FALSE;
   S486LH_CARTYPE.STN_Btype_1Arr[15] := FALSE;
   S486LH_CARTYPE.STN_Btype_2Arr[0] := FALSE;
   S486LH_CARTYPE.STN_Btype_2Arr[1] := FALSE;
   S486LH_CARTYPE.STN_Btype_2Arr[2] := FALSE;
   S486LH_CARTYPE.STN_Btype_2Arr[3] := FALSE;
   S486LH_CARTYPE.STN_Btype_2Arr[4] := FALSE;
   S486LH_CARTYPE.STN_Btype_2Arr[5] := FALSE;
   S486LH_CARTYPE.STN_Btype_2Arr[6] := FALSE;
   S486LH_CARTYPE.STN_Btype_2Arr[7] := FALSE;
   S486LH_CARTYPE.STN_Btype_2Arr[8] := FALSE;
   S486LH_CARTYPE.STN_Btype_2Arr[9] := FALSE;
   S486LH_CARTYPE.STN_Btype_2Arr[10] := FALSE;
   S486LH_CARTYPE.STN_Btype_2Arr[11] := FALSE;
   S486LH_CARTYPE.STN_Btype_2Arr[12] := FALSE;
   S486LH_CARTYPE.STN_Btype_2Arr[13] := FALSE;
   S486LH_CARTYPE.STN_Btype_2Arr[14] := FALSE;
   S486LH_CARTYPE.STN_Btype_2Arr[15] := FALSE;
   S486LH_CARTYPE.STN_Btype_3Arr[0] := FALSE;
   S486LH_CARTYPE.STN_Btype_3Arr[1] := FALSE;
   S486LH_CARTYPE.STN_Btype_3Arr[2] := FALSE;
   S486LH_CARTYPE.STN_Btype_3Arr[3] := FALSE;
   S486LH_CARTYPE.STN_Btype_3Arr[4] := FALSE;
   S486LH_CARTYPE.STN_Btype_3Arr[5] := FALSE;
   S486LH_CARTYPE.STN_Btype_3Arr[6] := FALSE;
   S486LH_CARTYPE.STN_Btype_3Arr[7] := FALSE;
   S486LH_CARTYPE.STN_Btype_3Arr[8] := FALSE;
   S486LH_CARTYPE.STN_Btype_3Arr[9] := FALSE;
   S486LH_CARTYPE.STN_Btype_3Arr[10] := FALSE;
   S486LH_CARTYPE.STN_Btype_3Arr[11] := FALSE;
   S486LH_CARTYPE.STN_Btype_3Arr[12] := FALSE;
   S486LH_CARTYPE.STN_Btype_3Arr[13] := FALSE;
   S486LH_CARTYPE.STN_Btype_3Arr[14] := FALSE;
   S486LH_CARTYPE.STN_Btype_3Arr[15] := FALSE;
   S486LH_CARTYPE.STN_Btype_4Arr[0] := FALSE;
   S486LH_CARTYPE.STN_Btype_4Arr[1] := FALSE;
   S486LH_CARTYPE.STN_Btype_4Arr[2] := FALSE;
   S486LH_CARTYPE.STN_Btype_4Arr[3] := FALSE;
   S486LH_CARTYPE.STN_Btype_4Arr[4] := FALSE;
   S486LH_CARTYPE.STN_Btype_4Arr[5] := FALSE;
   S486LH_CARTYPE.STN_Btype_4Arr[6] := FALSE;
   S486LH_CARTYPE.STN_Btype_4Arr[7] := FALSE;
   S486LH_CARTYPE.STN_Btype_4Arr[8] := FALSE;
   S486LH_CARTYPE.STN_Btype_4Arr[9] := FALSE;
   S486LH_CARTYPE.STN_Btype_4Arr[10] := FALSE;
   S486LH_CARTYPE.STN_Btype_4Arr[11] := FALSE;
   S486LH_CARTYPE.STN_Btype_4Arr[12] := FALSE;
   S486LH_CARTYPE.STN_Btype_4Arr[13] := FALSE;
   S486LH_CARTYPE.STN_Btype_4Arr[14] := FALSE;
   S486LH_CARTYPE.STN_Btype_4Arr[15] := FALSE;
   S486LH_CARTYPE.STN_Btype_5Arr[0] := FALSE;
   S486LH_CARTYPE.STN_Btype_5Arr[1] := FALSE;
   S486LH_CARTYPE.STN_Btype_5Arr[2] := FALSE;
   S486LH_CARTYPE.STN_Btype_5Arr[3] := FALSE;
   S486LH_CARTYPE.STN_Btype_5Arr[4] := FALSE;
   S486LH_CARTYPE.STN_Btype_5Arr[5] := FALSE;
   S486LH_CARTYPE.STN_Btype_5Arr[6] := FALSE;
   S486LH_CARTYPE.STN_Btype_5Arr[7] := FALSE;
   S486LH_CARTYPE.STN_Btype_5Arr[8] := FALSE;
   S486LH_CARTYPE.STN_Btype_5Arr[9] := FALSE;
   S486LH_CARTYPE.STN_Btype_5Arr[10] := FALSE;
   S486LH_CARTYPE.STN_Btype_5Arr[11] := FALSE;
   S486LH_CARTYPE.STN_Btype_5Arr[12] := FALSE;
   S486LH_CARTYPE.STN_Btype_5Arr[13] := FALSE;
   S486LH_CARTYPE.STN_Btype_5Arr[14] := FALSE;
   S486LH_CARTYPE.STN_Btype_5Arr[15] := FALSE;
   S486LH_CARTYPE.STN_Btype_6Arr[0] := FALSE;
   S486LH_CARTYPE.STN_Btype_6Arr[1] := FALSE;
   S486LH_CARTYPE.STN_Btype_6Arr[2] := FALSE;
   S486LH_CARTYPE.STN_Btype_6Arr[3] := FALSE;
   S486LH_CARTYPE.STN_Btype_6Arr[4] := FALSE;
   S486LH_CARTYPE.STN_Btype_6Arr[5] := FALSE;
   S486LH_CARTYPE.STN_Btype_6Arr[6] := FALSE;
   S486LH_CARTYPE.STN_Btype_6Arr[7] := FALSE;
   S486LH_CARTYPE.STN_Btype_6Arr[8] := FALSE;
   S486LH_CARTYPE.STN_Btype_6Arr[9] := FALSE;
   S486LH_CARTYPE.STN_Btype_6Arr[10] := FALSE;
   S486LH_CARTYPE.STN_Btype_6Arr[11] := FALSE;
   S486LH_CARTYPE.STN_Btype_6Arr[12] := FALSE;
   S486LH_CARTYPE.STN_Btype_6Arr[13] := FALSE;
   S486LH_CARTYPE.STN_Btype_6Arr[14] := FALSE;
   S486LH_CARTYPE.STN_Btype_6Arr[15] := FALSE;
   S486LH_CARTYPE.STN_1st_BT_On := FALSE;
   S486LH_CARTYPE.STN_2nd_BT_On := FALSE;
   S486LH_CARTYPE.STN_3rd_BT_On := FALSE;
   S486LH_CARTYPE.STN_4th_BT_On := FALSE;
   S486LH_CARTYPE.STN_5th_BT_On := FALSE;
   S486LH_CARTYPE.STN_6th_BT_On := FALSE;
   S486LH_CARTYPE.STN_7th_BT_On := FALSE;
   S486LH_CARTYPE.STN_8th_BT_On := FALSE;
   S486LH_CARTYPE.STN_9th_BT_On := FALSE;
   S486LH_CARTYPE.STN_10th_BT_On := FALSE;
   S486LH_CARTYPE.STN_11th_BT_On := FALSE;
   S486LH_CARTYPE.STN_12th_BT_On := FALSE;
   S486LH_CARTYPE.STN_1st_BT_Off := FALSE;
   S486LH_CARTYPE.BLKMove_Ret := 0;
   S486LH_CARTYPE.VIN_1BCD := W#16#0;
   S486LH_CARTYPE.VIN_2BCD := W#16#0;
   S486LH_CARTYPE.VIN_1Int := 0;
   S486LH_CARTYPE.VIN_2Int := 0;
   S711_CARTYPE.Stn_Vin_No := L#0;
   S711_CARTYPE.Stn_Bt_1Word := W#16#0;
   S711_CARTYPE.Stn_Bt_2Word := W#16#0;
   S711_CARTYPE.Stn_Bt_3Word := W#16#0;
   S711_CARTYPE.Stn_Bt_4Word := W#16#0;
   S711_CARTYPE.Stn_Bt_5Word_Sp := W#16#0;
   S711_CARTYPE.Stn_Bt_6Word_Sp := W#16#0;
   S711_CARTYPE.M_BType_On := FALSE;
   S711_CARTYPE.M_BType_None := FALSE;
   S711_CARTYPE.M_Bypass_BType := FALSE;
   S711_CARTYPE.M_BType_TL := FALSE;
   S711_CARTYPE.M_BType_LM := FALSE;
   S711_CARTYPE.M_BType_SP1 := FALSE;
   S711_CARTYPE.M_BType_SP2 := FALSE;
   S711_CARTYPE.M_BType_SP3 := FALSE;
   S711_CARTYPE.M_BType_DOM := FALSE;
   S711_CARTYPE.M_BType_EXP := FALSE;
   S711_CARTYPE.Robot_Prog_No := 0;
   S711_CARTYPE.STN_Btype_1Arr[0] := FALSE;
   S711_CARTYPE.STN_Btype_1Arr[1] := FALSE;
   S711_CARTYPE.STN_Btype_1Arr[2] := FALSE;
   S711_CARTYPE.STN_Btype_1Arr[3] := FALSE;
   S711_CARTYPE.STN_Btype_1Arr[4] := FALSE;
   S711_CARTYPE.STN_Btype_1Arr[5] := FALSE;
   S711_CARTYPE.STN_Btype_1Arr[6] := FALSE;
   S711_CARTYPE.STN_Btype_1Arr[7] := FALSE;
   S711_CARTYPE.STN_Btype_1Arr[8] := FALSE;
   S711_CARTYPE.STN_Btype_1Arr[9] := FALSE;
   S711_CARTYPE.STN_Btype_1Arr[10] := FALSE;
   S711_CARTYPE.STN_Btype_1Arr[11] := FALSE;
   S711_CARTYPE.STN_Btype_1Arr[12] := FALSE;
   S711_CARTYPE.STN_Btype_1Arr[13] := FALSE;
   S711_CARTYPE.STN_Btype_1Arr[14] := FALSE;
   S711_CARTYPE.STN_Btype_1Arr[15] := FALSE;
   S711_CARTYPE.STN_Btype_2Arr[0] := FALSE;
   S711_CARTYPE.STN_Btype_2Arr[1] := FALSE;
   S711_CARTYPE.STN_Btype_2Arr[2] := FALSE;
   S711_CARTYPE.STN_Btype_2Arr[3] := FALSE;
   S711_CARTYPE.STN_Btype_2Arr[4] := FALSE;
   S711_CARTYPE.STN_Btype_2Arr[5] := FALSE;
   S711_CARTYPE.STN_Btype_2Arr[6] := FALSE;
   S711_CARTYPE.STN_Btype_2Arr[7] := FALSE;
   S711_CARTYPE.STN_Btype_2Arr[8] := FALSE;
   S711_CARTYPE.STN_Btype_2Arr[9] := FALSE;
   S711_CARTYPE.STN_Btype_2Arr[10] := FALSE;
   S711_CARTYPE.STN_Btype_2Arr[11] := FALSE;
   S711_CARTYPE.STN_Btype_2Arr[12] := FALSE;
   S711_CARTYPE.STN_Btype_2Arr[13] := FALSE;
   S711_CARTYPE.STN_Btype_2Arr[14] := FALSE;
   S711_CARTYPE.STN_Btype_2Arr[15] := FALSE;
   S711_CARTYPE.STN_Btype_3Arr[0] := FALSE;
   S711_CARTYPE.STN_Btype_3Arr[1] := FALSE;
   S711_CARTYPE.STN_Btype_3Arr[2] := FALSE;
   S711_CARTYPE.STN_Btype_3Arr[3] := FALSE;
   S711_CARTYPE.STN_Btype_3Arr[4] := FALSE;
   S711_CARTYPE.STN_Btype_3Arr[5] := FALSE;
   S711_CARTYPE.STN_Btype_3Arr[6] := FALSE;
   S711_CARTYPE.STN_Btype_3Arr[7] := FALSE;
   S711_CARTYPE.STN_Btype_3Arr[8] := FALSE;
   S711_CARTYPE.STN_Btype_3Arr[9] := FALSE;
   S711_CARTYPE.STN_Btype_3Arr[10] := FALSE;
   S711_CARTYPE.STN_Btype_3Arr[11] := FALSE;
   S711_CARTYPE.STN_Btype_3Arr[12] := FALSE;
   S711_CARTYPE.STN_Btype_3Arr[13] := FALSE;
   S711_CARTYPE.STN_Btype_3Arr[14] := FALSE;
   S711_CARTYPE.STN_Btype_3Arr[15] := FALSE;
   S711_CARTYPE.STN_Btype_4Arr[0] := FALSE;
   S711_CARTYPE.STN_Btype_4Arr[1] := FALSE;
   S711_CARTYPE.STN_Btype_4Arr[2] := FALSE;
   S711_CARTYPE.STN_Btype_4Arr[3] := FALSE;
   S711_CARTYPE.STN_Btype_4Arr[4] := FALSE;
   S711_CARTYPE.STN_Btype_4Arr[5] := FALSE;
   S711_CARTYPE.STN_Btype_4Arr[6] := FALSE;
   S711_CARTYPE.STN_Btype_4Arr[7] := FALSE;
   S711_CARTYPE.STN_Btype_4Arr[8] := FALSE;
   S711_CARTYPE.STN_Btype_4Arr[9] := FALSE;
   S711_CARTYPE.STN_Btype_4Arr[10] := FALSE;
   S711_CARTYPE.STN_Btype_4Arr[11] := FALSE;
   S711_CARTYPE.STN_Btype_4Arr[12] := FALSE;
   S711_CARTYPE.STN_Btype_4Arr[13] := FALSE;
   S711_CARTYPE.STN_Btype_4Arr[14] := FALSE;
   S711_CARTYPE.STN_Btype_4Arr[15] := FALSE;
   S711_CARTYPE.STN_Btype_5Arr[0] := FALSE;
   S711_CARTYPE.STN_Btype_5Arr[1] := FALSE;
   S711_CARTYPE.STN_Btype_5Arr[2] := FALSE;
   S711_CARTYPE.STN_Btype_5Arr[3] := FALSE;
   S711_CARTYPE.STN_Btype_5Arr[4] := FALSE;
   S711_CARTYPE.STN_Btype_5Arr[5] := FALSE;
   S711_CARTYPE.STN_Btype_5Arr[6] := FALSE;
   S711_CARTYPE.STN_Btype_5Arr[7] := FALSE;
   S711_CARTYPE.STN_Btype_5Arr[8] := FALSE;
   S711_CARTYPE.STN_Btype_5Arr[9] := FALSE;
   S711_CARTYPE.STN_Btype_5Arr[10] := FALSE;
   S711_CARTYPE.STN_Btype_5Arr[11] := FALSE;
   S711_CARTYPE.STN_Btype_5Arr[12] := FALSE;
   S711_CARTYPE.STN_Btype_5Arr[13] := FALSE;
   S711_CARTYPE.STN_Btype_5Arr[14] := FALSE;
   S711_CARTYPE.STN_Btype_5Arr[15] := FALSE;
   S711_CARTYPE.STN_Btype_6Arr[0] := FALSE;
   S711_CARTYPE.STN_Btype_6Arr[1] := FALSE;
   S711_CARTYPE.STN_Btype_6Arr[2] := FALSE;
   S711_CARTYPE.STN_Btype_6Arr[3] := FALSE;
   S711_CARTYPE.STN_Btype_6Arr[4] := FALSE;
   S711_CARTYPE.STN_Btype_6Arr[5] := FALSE;
   S711_CARTYPE.STN_Btype_6Arr[6] := FALSE;
   S711_CARTYPE.STN_Btype_6Arr[7] := FALSE;
   S711_CARTYPE.STN_Btype_6Arr[8] := FALSE;
   S711_CARTYPE.STN_Btype_6Arr[9] := FALSE;
   S711_CARTYPE.STN_Btype_6Arr[10] := FALSE;
   S711_CARTYPE.STN_Btype_6Arr[11] := FALSE;
   S711_CARTYPE.STN_Btype_6Arr[12] := FALSE;
   S711_CARTYPE.STN_Btype_6Arr[13] := FALSE;
   S711_CARTYPE.STN_Btype_6Arr[14] := FALSE;
   S711_CARTYPE.STN_Btype_6Arr[15] := FALSE;
   S711_CARTYPE.STN_1st_BT_On := FALSE;
   S711_CARTYPE.STN_2nd_BT_On := FALSE;
   S711_CARTYPE.STN_3rd_BT_On := FALSE;
   S711_CARTYPE.STN_4th_BT_On := FALSE;
   S711_CARTYPE.STN_5th_BT_On := FALSE;
   S711_CARTYPE.STN_6th_BT_On := FALSE;
   S711_CARTYPE.STN_7th_BT_On := FALSE;
   S711_CARTYPE.STN_8th_BT_On := FALSE;
   S711_CARTYPE.STN_9th_BT_On := FALSE;
   S711_CARTYPE.STN_10th_BT_On := FALSE;
   S711_CARTYPE.STN_11th_BT_On := FALSE;
   S711_CARTYPE.STN_12th_BT_On := FALSE;
   S711_CARTYPE.STN_1st_BT_Off := FALSE;
   S711_CARTYPE.BLKMove_Ret := 0;
   S711_CARTYPE.VIN_1BCD := W#16#0;
   S711_CARTYPE.VIN_2BCD := W#16#0;
   S711_CARTYPE.VIN_1Int := 0;
   S711_CARTYPE.VIN_2Int := 0;
   S711R1_R2_CARTYPE.Stn_Vin_No := L#0;
   S711R1_R2_CARTYPE.Stn_Bt_1Word := W#16#0;
   S711R1_R2_CARTYPE.Stn_Bt_2Word := W#16#0;
   S711R1_R2_CARTYPE.Stn_Bt_3Word := W#16#0;
   S711R1_R2_CARTYPE.Stn_Bt_4Word := W#16#0;
   S711R1_R2_CARTYPE.Stn_Bt_5Word_Sp := W#16#0;
   S711R1_R2_CARTYPE.Stn_Bt_6Word_Sp := W#16#0;
   S711R1_R2_CARTYPE.M_BType_On := FALSE;
   S711R1_R2_CARTYPE.M_BType_None := FALSE;
   S711R1_R2_CARTYPE.M_Bypass_BType := FALSE;
   S711R1_R2_CARTYPE.M_BType_TL := FALSE;
   S711R1_R2_CARTYPE.M_BType_LM := FALSE;
   S711R1_R2_CARTYPE.M_BType_SP1 := FALSE;
   S711R1_R2_CARTYPE.M_BType_SP2 := FALSE;
   S711R1_R2_CARTYPE.M_BType_SP3 := FALSE;
   S711R1_R2_CARTYPE.M_BType_DOM := FALSE;
   S711R1_R2_CARTYPE.M_BType_EXP := FALSE;
   S711R1_R2_CARTYPE.Robot_Prog_No := 0;
   S711R1_R2_CARTYPE.STN_Btype_1Arr[0] := FALSE;
   S711R1_R2_CARTYPE.STN_Btype_1Arr[1] := FALSE;
   S711R1_R2_CARTYPE.STN_Btype_1Arr[2] := FALSE;
   S711R1_R2_CARTYPE.STN_Btype_1Arr[3] := FALSE;
   S711R1_R2_CARTYPE.STN_Btype_1Arr[4] := FALSE;
   S711R1_R2_CARTYPE.STN_Btype_1Arr[5] := FALSE;
   S711R1_R2_CARTYPE.STN_Btype_1Arr[6] := FALSE;
   S711R1_R2_CARTYPE.STN_Btype_1Arr[7] := FALSE;
   S711R1_R2_CARTYPE.STN_Btype_1Arr[8] := FALSE;
   S711R1_R2_CARTYPE.STN_Btype_1Arr[9] := FALSE;
   S711R1_R2_CARTYPE.STN_Btype_1Arr[10] := FALSE;
   S711R1_R2_CARTYPE.STN_Btype_1Arr[11] := FALSE;
   S711R1_R2_CARTYPE.STN_Btype_1Arr[12] := FALSE;
   S711R1_R2_CARTYPE.STN_Btype_1Arr[13] := FALSE;
   S711R1_R2_CARTYPE.STN_Btype_1Arr[14] := FALSE;
   S711R1_R2_CARTYPE.STN_Btype_1Arr[15] := FALSE;
   S711R1_R2_CARTYPE.STN_Btype_2Arr[0] := FALSE;
   S711R1_R2_CARTYPE.STN_Btype_2Arr[1] := FALSE;
   S711R1_R2_CARTYPE.STN_Btype_2Arr[2] := FALSE;
   S711R1_R2_CARTYPE.STN_Btype_2Arr[3] := FALSE;
   S711R1_R2_CARTYPE.STN_Btype_2Arr[4] := FALSE;
   S711R1_R2_CARTYPE.STN_Btype_2Arr[5] := FALSE;
   S711R1_R2_CARTYPE.STN_Btype_2Arr[6] := FALSE;
   S711R1_R2_CARTYPE.STN_Btype_2Arr[7] := FALSE;
   S711R1_R2_CARTYPE.STN_Btype_2Arr[8] := FALSE;
   S711R1_R2_CARTYPE.STN_Btype_2Arr[9] := FALSE;
   S711R1_R2_CARTYPE.STN_Btype_2Arr[10] := FALSE;
   S711R1_R2_CARTYPE.STN_Btype_2Arr[11] := FALSE;
   S711R1_R2_CARTYPE.STN_Btype_2Arr[12] := FALSE;
   S711R1_R2_CARTYPE.STN_Btype_2Arr[13] := FALSE;
   S711R1_R2_CARTYPE.STN_Btype_2Arr[14] := FALSE;
   S711R1_R2_CARTYPE.STN_Btype_2Arr[15] := FALSE;
   S711R1_R2_CARTYPE.STN_Btype_3Arr[0] := FALSE;
   S711R1_R2_CARTYPE.STN_Btype_3Arr[1] := FALSE;
   S711R1_R2_CARTYPE.STN_Btype_3Arr[2] := FALSE;
   S711R1_R2_CARTYPE.STN_Btype_3Arr[3] := FALSE;
   S711R1_R2_CARTYPE.STN_Btype_3Arr[4] := FALSE;
   S711R1_R2_CARTYPE.STN_Btype_3Arr[5] := FALSE;
   S711R1_R2_CARTYPE.STN_Btype_3Arr[6] := FALSE;
   S711R1_R2_CARTYPE.STN_Btype_3Arr[7] := FALSE;
   S711R1_R2_CARTYPE.STN_Btype_3Arr[8] := FALSE;
   S711R1_R2_CARTYPE.STN_Btype_3Arr[9] := FALSE;
   S711R1_R2_CARTYPE.STN_Btype_3Arr[10] := FALSE;
   S711R1_R2_CARTYPE.STN_Btype_3Arr[11] := FALSE;
   S711R1_R2_CARTYPE.STN_Btype_3Arr[12] := FALSE;
   S711R1_R2_CARTYPE.STN_Btype_3Arr[13] := FALSE;
   S711R1_R2_CARTYPE.STN_Btype_3Arr[14] := FALSE;
   S711R1_R2_CARTYPE.STN_Btype_3Arr[15] := FALSE;
   S711R1_R2_CARTYPE.STN_Btype_4Arr[0] := FALSE;
   S711R1_R2_CARTYPE.STN_Btype_4Arr[1] := FALSE;
   S711R1_R2_CARTYPE.STN_Btype_4Arr[2] := FALSE;
   S711R1_R2_CARTYPE.STN_Btype_4Arr[3] := FALSE;
   S711R1_R2_CARTYPE.STN_Btype_4Arr[4] := FALSE;
   S711R1_R2_CARTYPE.STN_Btype_4Arr[5] := FALSE;
   S711R1_R2_CARTYPE.STN_Btype_4Arr[6] := FALSE;
   S711R1_R2_CARTYPE.STN_Btype_4Arr[7] := FALSE;
   S711R1_R2_CARTYPE.STN_Btype_4Arr[8] := FALSE;
   S711R1_R2_CARTYPE.STN_Btype_4Arr[9] := FALSE;
   S711R1_R2_CARTYPE.STN_Btype_4Arr[10] := FALSE;
   S711R1_R2_CARTYPE.STN_Btype_4Arr[11] := FALSE;
   S711R1_R2_CARTYPE.STN_Btype_4Arr[12] := FALSE;
   S711R1_R2_CARTYPE.STN_Btype_4Arr[13] := FALSE;
   S711R1_R2_CARTYPE.STN_Btype_4Arr[14] := FALSE;
   S711R1_R2_CARTYPE.STN_Btype_4Arr[15] := FALSE;
   S711R1_R2_CARTYPE.STN_Btype_5Arr[0] := FALSE;
   S711R1_R2_CARTYPE.STN_Btype_5Arr[1] := FALSE;
   S711R1_R2_CARTYPE.STN_Btype_5Arr[2] := FALSE;
   S711R1_R2_CARTYPE.STN_Btype_5Arr[3] := FALSE;
   S711R1_R2_CARTYPE.STN_Btype_5Arr[4] := FALSE;
   S711R1_R2_CARTYPE.STN_Btype_5Arr[5] := FALSE;
   S711R1_R2_CARTYPE.STN_Btype_5Arr[6] := FALSE;
   S711R1_R2_CARTYPE.STN_Btype_5Arr[7] := FALSE;
   S711R1_R2_CARTYPE.STN_Btype_5Arr[8] := FALSE;
   S711R1_R2_CARTYPE.STN_Btype_5Arr[9] := FALSE;
   S711R1_R2_CARTYPE.STN_Btype_5Arr[10] := FALSE;
   S711R1_R2_CARTYPE.STN_Btype_5Arr[11] := FALSE;
   S711R1_R2_CARTYPE.STN_Btype_5Arr[12] := FALSE;
   S711R1_R2_CARTYPE.STN_Btype_5Arr[13] := FALSE;
   S711R1_R2_CARTYPE.STN_Btype_5Arr[14] := FALSE;
   S711R1_R2_CARTYPE.STN_Btype_5Arr[15] := FALSE;
   S711R1_R2_CARTYPE.STN_Btype_6Arr[0] := FALSE;
   S711R1_R2_CARTYPE.STN_Btype_6Arr[1] := FALSE;
   S711R1_R2_CARTYPE.STN_Btype_6Arr[2] := FALSE;
   S711R1_R2_CARTYPE.STN_Btype_6Arr[3] := FALSE;
   S711R1_R2_CARTYPE.STN_Btype_6Arr[4] := FALSE;
   S711R1_R2_CARTYPE.STN_Btype_6Arr[5] := FALSE;
   S711R1_R2_CARTYPE.STN_Btype_6Arr[6] := FALSE;
   S711R1_R2_CARTYPE.STN_Btype_6Arr[7] := FALSE;
   S711R1_R2_CARTYPE.STN_Btype_6Arr[8] := FALSE;
   S711R1_R2_CARTYPE.STN_Btype_6Arr[9] := FALSE;
   S711R1_R2_CARTYPE.STN_Btype_6Arr[10] := FALSE;
   S711R1_R2_CARTYPE.STN_Btype_6Arr[11] := FALSE;
   S711R1_R2_CARTYPE.STN_Btype_6Arr[12] := FALSE;
   S711R1_R2_CARTYPE.STN_Btype_6Arr[13] := FALSE;
   S711R1_R2_CARTYPE.STN_Btype_6Arr[14] := FALSE;
   S711R1_R2_CARTYPE.STN_Btype_6Arr[15] := FALSE;
   S711R1_R2_CARTYPE.STN_1st_BT_On := FALSE;
   S711R1_R2_CARTYPE.STN_2nd_BT_On := FALSE;
   S711R1_R2_CARTYPE.STN_3rd_BT_On := FALSE;
   S711R1_R2_CARTYPE.STN_4th_BT_On := FALSE;
   S711R1_R2_CARTYPE.STN_5th_BT_On := FALSE;
   S711R1_R2_CARTYPE.STN_6th_BT_On := FALSE;
   S711R1_R2_CARTYPE.STN_7th_BT_On := FALSE;
   S711R1_R2_CARTYPE.STN_8th_BT_On := FALSE;
   S711R1_R2_CARTYPE.STN_9th_BT_On := FALSE;
   S711R1_R2_CARTYPE.STN_10th_BT_On := FALSE;
   S711R1_R2_CARTYPE.STN_11th_BT_On := FALSE;
   S711R1_R2_CARTYPE.STN_12th_BT_On := FALSE;
   S711R1_R2_CARTYPE.STN_1st_BT_Off := FALSE;
   S711R1_R2_CARTYPE.BLKMove_Ret := 0;
   S711R1_R2_CARTYPE.VIN_1BCD := W#16#0;
   S711R1_R2_CARTYPE.VIN_2BCD := W#16#0;
   S711R1_R2_CARTYPE.VIN_1Int := 0;
   S711R1_R2_CARTYPE.VIN_2Int := 0;
   S711A_FAC_CARTYPE.Stn_Vin_No := L#0;
   S711A_FAC_CARTYPE.Stn_Bt_1Word := W#16#0;
   S711A_FAC_CARTYPE.Stn_Bt_2Word := W#16#0;
   S711A_FAC_CARTYPE.Stn_Bt_3Word := W#16#0;
   S711A_FAC_CARTYPE.Stn_Bt_4Word := W#16#0;
   S711A_FAC_CARTYPE.Stn_Bt_5Word_Sp := W#16#0;
   S711A_FAC_CARTYPE.Stn_Bt_6Word_Sp := W#16#0;
   S711A_FAC_CARTYPE.M_BType_On := FALSE;
   S711A_FAC_CARTYPE.M_BType_None := FALSE;
   S711A_FAC_CARTYPE.M_Bypass_BType := FALSE;
   S711A_FAC_CARTYPE.M_BType_TL := FALSE;
   S711A_FAC_CARTYPE.M_BType_LM := FALSE;
   S711A_FAC_CARTYPE.M_BType_SP1 := FALSE;
   S711A_FAC_CARTYPE.M_BType_SP2 := FALSE;
   S711A_FAC_CARTYPE.M_BType_SP3 := FALSE;
   S711A_FAC_CARTYPE.M_BType_DOM := FALSE;
   S711A_FAC_CARTYPE.M_BType_EXP := FALSE;
   S711A_FAC_CARTYPE.Robot_Prog_No := 0;
   S711A_FAC_CARTYPE.STN_Btype_1Arr[0] := FALSE;
   S711A_FAC_CARTYPE.STN_Btype_1Arr[1] := FALSE;
   S711A_FAC_CARTYPE.STN_Btype_1Arr[2] := FALSE;
   S711A_FAC_CARTYPE.STN_Btype_1Arr[3] := FALSE;
   S711A_FAC_CARTYPE.STN_Btype_1Arr[4] := FALSE;
   S711A_FAC_CARTYPE.STN_Btype_1Arr[5] := FALSE;
   S711A_FAC_CARTYPE.STN_Btype_1Arr[6] := FALSE;
   S711A_FAC_CARTYPE.STN_Btype_1Arr[7] := FALSE;
   S711A_FAC_CARTYPE.STN_Btype_1Arr[8] := FALSE;
   S711A_FAC_CARTYPE.STN_Btype_1Arr[9] := FALSE;
   S711A_FAC_CARTYPE.STN_Btype_1Arr[10] := FALSE;
   S711A_FAC_CARTYPE.STN_Btype_1Arr[11] := FALSE;
   S711A_FAC_CARTYPE.STN_Btype_1Arr[12] := FALSE;
   S711A_FAC_CARTYPE.STN_Btype_1Arr[13] := FALSE;
   S711A_FAC_CARTYPE.STN_Btype_1Arr[14] := FALSE;
   S711A_FAC_CARTYPE.STN_Btype_1Arr[15] := FALSE;
   S711A_FAC_CARTYPE.STN_Btype_2Arr[0] := FALSE;
   S711A_FAC_CARTYPE.STN_Btype_2Arr[1] := FALSE;
   S711A_FAC_CARTYPE.STN_Btype_2Arr[2] := FALSE;
   S711A_FAC_CARTYPE.STN_Btype_2Arr[3] := FALSE;
   S711A_FAC_CARTYPE.STN_Btype_2Arr[4] := FALSE;
   S711A_FAC_CARTYPE.STN_Btype_2Arr[5] := FALSE;
   S711A_FAC_CARTYPE.STN_Btype_2Arr[6] := FALSE;
   S711A_FAC_CARTYPE.STN_Btype_2Arr[7] := FALSE;
   S711A_FAC_CARTYPE.STN_Btype_2Arr[8] := FALSE;
   S711A_FAC_CARTYPE.STN_Btype_2Arr[9] := FALSE;
   S711A_FAC_CARTYPE.STN_Btype_2Arr[10] := FALSE;
   S711A_FAC_CARTYPE.STN_Btype_2Arr[11] := FALSE;
   S711A_FAC_CARTYPE.STN_Btype_2Arr[12] := FALSE;
   S711A_FAC_CARTYPE.STN_Btype_2Arr[13] := FALSE;
   S711A_FAC_CARTYPE.STN_Btype_2Arr[14] := FALSE;
   S711A_FAC_CARTYPE.STN_Btype_2Arr[15] := FALSE;
   S711A_FAC_CARTYPE.STN_Btype_3Arr[0] := FALSE;
   S711A_FAC_CARTYPE.STN_Btype_3Arr[1] := FALSE;
   S711A_FAC_CARTYPE.STN_Btype_3Arr[2] := FALSE;
   S711A_FAC_CARTYPE.STN_Btype_3Arr[3] := FALSE;
   S711A_FAC_CARTYPE.STN_Btype_3Arr[4] := FALSE;
   S711A_FAC_CARTYPE.STN_Btype_3Arr[5] := FALSE;
   S711A_FAC_CARTYPE.STN_Btype_3Arr[6] := FALSE;
   S711A_FAC_CARTYPE.STN_Btype_3Arr[7] := FALSE;
   S711A_FAC_CARTYPE.STN_Btype_3Arr[8] := FALSE;
   S711A_FAC_CARTYPE.STN_Btype_3Arr[9] := FALSE;
   S711A_FAC_CARTYPE.STN_Btype_3Arr[10] := FALSE;
   S711A_FAC_CARTYPE.STN_Btype_3Arr[11] := FALSE;
   S711A_FAC_CARTYPE.STN_Btype_3Arr[12] := FALSE;
   S711A_FAC_CARTYPE.STN_Btype_3Arr[13] := FALSE;
   S711A_FAC_CARTYPE.STN_Btype_3Arr[14] := FALSE;
   S711A_FAC_CARTYPE.STN_Btype_3Arr[15] := FALSE;
   S711A_FAC_CARTYPE.STN_Btype_4Arr[0] := FALSE;
   S711A_FAC_CARTYPE.STN_Btype_4Arr[1] := FALSE;
   S711A_FAC_CARTYPE.STN_Btype_4Arr[2] := FALSE;
   S711A_FAC_CARTYPE.STN_Btype_4Arr[3] := FALSE;
   S711A_FAC_CARTYPE.STN_Btype_4Arr[4] := FALSE;
   S711A_FAC_CARTYPE.STN_Btype_4Arr[5] := FALSE;
   S711A_FAC_CARTYPE.STN_Btype_4Arr[6] := FALSE;
   S711A_FAC_CARTYPE.STN_Btype_4Arr[7] := FALSE;
   S711A_FAC_CARTYPE.STN_Btype_4Arr[8] := FALSE;
   S711A_FAC_CARTYPE.STN_Btype_4Arr[9] := FALSE;
   S711A_FAC_CARTYPE.STN_Btype_4Arr[10] := FALSE;
   S711A_FAC_CARTYPE.STN_Btype_4Arr[11] := FALSE;
   S711A_FAC_CARTYPE.STN_Btype_4Arr[12] := FALSE;
   S711A_FAC_CARTYPE.STN_Btype_4Arr[13] := FALSE;
   S711A_FAC_CARTYPE.STN_Btype_4Arr[14] := FALSE;
   S711A_FAC_CARTYPE.STN_Btype_4Arr[15] := FALSE;
   S711A_FAC_CARTYPE.STN_Btype_5Arr[0] := FALSE;
   S711A_FAC_CARTYPE.STN_Btype_5Arr[1] := FALSE;
   S711A_FAC_CARTYPE.STN_Btype_5Arr[2] := FALSE;
   S711A_FAC_CARTYPE.STN_Btype_5Arr[3] := FALSE;
   S711A_FAC_CARTYPE.STN_Btype_5Arr[4] := FALSE;
   S711A_FAC_CARTYPE.STN_Btype_5Arr[5] := FALSE;
   S711A_FAC_CARTYPE.STN_Btype_5Arr[6] := FALSE;
   S711A_FAC_CARTYPE.STN_Btype_5Arr[7] := FALSE;
   S711A_FAC_CARTYPE.STN_Btype_5Arr[8] := FALSE;
   S711A_FAC_CARTYPE.STN_Btype_5Arr[9] := FALSE;
   S711A_FAC_CARTYPE.STN_Btype_5Arr[10] := FALSE;
   S711A_FAC_CARTYPE.STN_Btype_5Arr[11] := FALSE;
   S711A_FAC_CARTYPE.STN_Btype_5Arr[12] := FALSE;
   S711A_FAC_CARTYPE.STN_Btype_5Arr[13] := FALSE;
   S711A_FAC_CARTYPE.STN_Btype_5Arr[14] := FALSE;
   S711A_FAC_CARTYPE.STN_Btype_5Arr[15] := FALSE;
   S711A_FAC_CARTYPE.STN_Btype_6Arr[0] := FALSE;
   S711A_FAC_CARTYPE.STN_Btype_6Arr[1] := FALSE;
   S711A_FAC_CARTYPE.STN_Btype_6Arr[2] := FALSE;
   S711A_FAC_CARTYPE.STN_Btype_6Arr[3] := FALSE;
   S711A_FAC_CARTYPE.STN_Btype_6Arr[4] := FALSE;
   S711A_FAC_CARTYPE.STN_Btype_6Arr[5] := FALSE;
   S711A_FAC_CARTYPE.STN_Btype_6Arr[6] := FALSE;
   S711A_FAC_CARTYPE.STN_Btype_6Arr[7] := FALSE;
   S711A_FAC_CARTYPE.STN_Btype_6Arr[8] := FALSE;
   S711A_FAC_CARTYPE.STN_Btype_6Arr[9] := FALSE;
   S711A_FAC_CARTYPE.STN_Btype_6Arr[10] := FALSE;
   S711A_FAC_CARTYPE.STN_Btype_6Arr[11] := FALSE;
   S711A_FAC_CARTYPE.STN_Btype_6Arr[12] := FALSE;
   S711A_FAC_CARTYPE.STN_Btype_6Arr[13] := FALSE;
   S711A_FAC_CARTYPE.STN_Btype_6Arr[14] := FALSE;
   S711A_FAC_CARTYPE.STN_Btype_6Arr[15] := FALSE;
   S711A_FAC_CARTYPE.STN_1st_BT_On := FALSE;
   S711A_FAC_CARTYPE.STN_2nd_BT_On := FALSE;
   S711A_FAC_CARTYPE.STN_3rd_BT_On := FALSE;
   S711A_FAC_CARTYPE.STN_4th_BT_On := FALSE;
   S711A_FAC_CARTYPE.STN_5th_BT_On := FALSE;
   S711A_FAC_CARTYPE.STN_6th_BT_On := FALSE;
   S711A_FAC_CARTYPE.STN_7th_BT_On := FALSE;
   S711A_FAC_CARTYPE.STN_8th_BT_On := FALSE;
   S711A_FAC_CARTYPE.STN_9th_BT_On := FALSE;
   S711A_FAC_CARTYPE.STN_10th_BT_On := FALSE;
   S711A_FAC_CARTYPE.STN_11th_BT_On := FALSE;
   S711A_FAC_CARTYPE.STN_12th_BT_On := FALSE;
   S711A_FAC_CARTYPE.STN_1st_BT_Off := FALSE;
   S711A_FAC_CARTYPE.BLKMove_Ret := 0;
   S711A_FAC_CARTYPE.VIN_1BCD := W#16#0;
   S711A_FAC_CARTYPE.VIN_2BCD := W#16#0;
   S711A_FAC_CARTYPE.VIN_1Int := 0;
   S711A_FAC_CARTYPE.VIN_2Int := 0;
   S711AB_KEY_CARTYPE.Stn_Vin_No := L#0;
   S711AB_KEY_CARTYPE.Stn_Bt_1Word := W#16#0;
   S711AB_KEY_CARTYPE.Stn_Bt_2Word := W#16#0;
   S711AB_KEY_CARTYPE.Stn_Bt_3Word := W#16#0;
   S711AB_KEY_CARTYPE.Stn_Bt_4Word := W#16#0;
   S711AB_KEY_CARTYPE.Stn_Bt_5Word_Sp := W#16#0;
   S711AB_KEY_CARTYPE.Stn_Bt_6Word_Sp := W#16#0;
   S711AB_KEY_CARTYPE.M_BType_On := FALSE;
   S711AB_KEY_CARTYPE.M_BType_None := FALSE;
   S711AB_KEY_CARTYPE.M_Bypass_BType := FALSE;
   S711AB_KEY_CARTYPE.M_BType_TL := FALSE;
   S711AB_KEY_CARTYPE.M_BType_LM := FALSE;
   S711AB_KEY_CARTYPE.M_BType_SP1 := FALSE;
   S711AB_KEY_CARTYPE.M_BType_SP2 := FALSE;
   S711AB_KEY_CARTYPE.M_BType_SP3 := FALSE;
   S711AB_KEY_CARTYPE.M_BType_DOM := FALSE;
   S711AB_KEY_CARTYPE.M_BType_EXP := FALSE;
   S711AB_KEY_CARTYPE.Robot_Prog_No := 0;
   S711AB_KEY_CARTYPE.STN_Btype_1Arr[0] := FALSE;
   S711AB_KEY_CARTYPE.STN_Btype_1Arr[1] := FALSE;
   S711AB_KEY_CARTYPE.STN_Btype_1Arr[2] := FALSE;
   S711AB_KEY_CARTYPE.STN_Btype_1Arr[3] := FALSE;
   S711AB_KEY_CARTYPE.STN_Btype_1Arr[4] := FALSE;
   S711AB_KEY_CARTYPE.STN_Btype_1Arr[5] := FALSE;
   S711AB_KEY_CARTYPE.STN_Btype_1Arr[6] := FALSE;
   S711AB_KEY_CARTYPE.STN_Btype_1Arr[7] := FALSE;
   S711AB_KEY_CARTYPE.STN_Btype_1Arr[8] := FALSE;
   S711AB_KEY_CARTYPE.STN_Btype_1Arr[9] := FALSE;
   S711AB_KEY_CARTYPE.STN_Btype_1Arr[10] := FALSE;
   S711AB_KEY_CARTYPE.STN_Btype_1Arr[11] := FALSE;
   S711AB_KEY_CARTYPE.STN_Btype_1Arr[12] := FALSE;
   S711AB_KEY_CARTYPE.STN_Btype_1Arr[13] := FALSE;
   S711AB_KEY_CARTYPE.STN_Btype_1Arr[14] := FALSE;
   S711AB_KEY_CARTYPE.STN_Btype_1Arr[15] := FALSE;
   S711AB_KEY_CARTYPE.STN_Btype_2Arr[0] := FALSE;
   S711AB_KEY_CARTYPE.STN_Btype_2Arr[1] := FALSE;
   S711AB_KEY_CARTYPE.STN_Btype_2Arr[2] := FALSE;
   S711AB_KEY_CARTYPE.STN_Btype_2Arr[3] := FALSE;
   S711AB_KEY_CARTYPE.STN_Btype_2Arr[4] := FALSE;
   S711AB_KEY_CARTYPE.STN_Btype_2Arr[5] := FALSE;
   S711AB_KEY_CARTYPE.STN_Btype_2Arr[6] := FALSE;
   S711AB_KEY_CARTYPE.STN_Btype_2Arr[7] := FALSE;
   S711AB_KEY_CARTYPE.STN_Btype_2Arr[8] := FALSE;
   S711AB_KEY_CARTYPE.STN_Btype_2Arr[9] := FALSE;
   S711AB_KEY_CARTYPE.STN_Btype_2Arr[10] := FALSE;
   S711AB_KEY_CARTYPE.STN_Btype_2Arr[11] := FALSE;
   S711AB_KEY_CARTYPE.STN_Btype_2Arr[12] := FALSE;
   S711AB_KEY_CARTYPE.STN_Btype_2Arr[13] := FALSE;
   S711AB_KEY_CARTYPE.STN_Btype_2Arr[14] := FALSE;
   S711AB_KEY_CARTYPE.STN_Btype_2Arr[15] := FALSE;
   S711AB_KEY_CARTYPE.STN_Btype_3Arr[0] := FALSE;
   S711AB_KEY_CARTYPE.STN_Btype_3Arr[1] := FALSE;
   S711AB_KEY_CARTYPE.STN_Btype_3Arr[2] := FALSE;
   S711AB_KEY_CARTYPE.STN_Btype_3Arr[3] := FALSE;
   S711AB_KEY_CARTYPE.STN_Btype_3Arr[4] := FALSE;
   S711AB_KEY_CARTYPE.STN_Btype_3Arr[5] := FALSE;
   S711AB_KEY_CARTYPE.STN_Btype_3Arr[6] := FALSE;
   S711AB_KEY_CARTYPE.STN_Btype_3Arr[7] := FALSE;
   S711AB_KEY_CARTYPE.STN_Btype_3Arr[8] := FALSE;
   S711AB_KEY_CARTYPE.STN_Btype_3Arr[9] := FALSE;
   S711AB_KEY_CARTYPE.STN_Btype_3Arr[10] := FALSE;
   S711AB_KEY_CARTYPE.STN_Btype_3Arr[11] := FALSE;
   S711AB_KEY_CARTYPE.STN_Btype_3Arr[12] := FALSE;
   S711AB_KEY_CARTYPE.STN_Btype_3Arr[13] := FALSE;
   S711AB_KEY_CARTYPE.STN_Btype_3Arr[14] := FALSE;
   S711AB_KEY_CARTYPE.STN_Btype_3Arr[15] := FALSE;
   S711AB_KEY_CARTYPE.STN_Btype_4Arr[0] := FALSE;
   S711AB_KEY_CARTYPE.STN_Btype_4Arr[1] := FALSE;
   S711AB_KEY_CARTYPE.STN_Btype_4Arr[2] := FALSE;
   S711AB_KEY_CARTYPE.STN_Btype_4Arr[3] := FALSE;
   S711AB_KEY_CARTYPE.STN_Btype_4Arr[4] := FALSE;
   S711AB_KEY_CARTYPE.STN_Btype_4Arr[5] := FALSE;
   S711AB_KEY_CARTYPE.STN_Btype_4Arr[6] := FALSE;
   S711AB_KEY_CARTYPE.STN_Btype_4Arr[7] := FALSE;
   S711AB_KEY_CARTYPE.STN_Btype_4Arr[8] := FALSE;
   S711AB_KEY_CARTYPE.STN_Btype_4Arr[9] := FALSE;
   S711AB_KEY_CARTYPE.STN_Btype_4Arr[10] := FALSE;
   S711AB_KEY_CARTYPE.STN_Btype_4Arr[11] := FALSE;
   S711AB_KEY_CARTYPE.STN_Btype_4Arr[12] := FALSE;
   S711AB_KEY_CARTYPE.STN_Btype_4Arr[13] := FALSE;
   S711AB_KEY_CARTYPE.STN_Btype_4Arr[14] := FALSE;
   S711AB_KEY_CARTYPE.STN_Btype_4Arr[15] := FALSE;
   S711AB_KEY_CARTYPE.STN_Btype_5Arr[0] := FALSE;
   S711AB_KEY_CARTYPE.STN_Btype_5Arr[1] := FALSE;
   S711AB_KEY_CARTYPE.STN_Btype_5Arr[2] := FALSE;
   S711AB_KEY_CARTYPE.STN_Btype_5Arr[3] := FALSE;
   S711AB_KEY_CARTYPE.STN_Btype_5Arr[4] := FALSE;
   S711AB_KEY_CARTYPE.STN_Btype_5Arr[5] := FALSE;
   S711AB_KEY_CARTYPE.STN_Btype_5Arr[6] := FALSE;
   S711AB_KEY_CARTYPE.STN_Btype_5Arr[7] := FALSE;
   S711AB_KEY_CARTYPE.STN_Btype_5Arr[8] := FALSE;
   S711AB_KEY_CARTYPE.STN_Btype_5Arr[9] := FALSE;
   S711AB_KEY_CARTYPE.STN_Btype_5Arr[10] := FALSE;
   S711AB_KEY_CARTYPE.STN_Btype_5Arr[11] := FALSE;
   S711AB_KEY_CARTYPE.STN_Btype_5Arr[12] := FALSE;
   S711AB_KEY_CARTYPE.STN_Btype_5Arr[13] := FALSE;
   S711AB_KEY_CARTYPE.STN_Btype_5Arr[14] := FALSE;
   S711AB_KEY_CARTYPE.STN_Btype_5Arr[15] := FALSE;
   S711AB_KEY_CARTYPE.STN_Btype_6Arr[0] := FALSE;
   S711AB_KEY_CARTYPE.STN_Btype_6Arr[1] := FALSE;
   S711AB_KEY_CARTYPE.STN_Btype_6Arr[2] := FALSE;
   S711AB_KEY_CARTYPE.STN_Btype_6Arr[3] := FALSE;
   S711AB_KEY_CARTYPE.STN_Btype_6Arr[4] := FALSE;
   S711AB_KEY_CARTYPE.STN_Btype_6Arr[5] := FALSE;
   S711AB_KEY_CARTYPE.STN_Btype_6Arr[6] := FALSE;
   S711AB_KEY_CARTYPE.STN_Btype_6Arr[7] := FALSE;
   S711AB_KEY_CARTYPE.STN_Btype_6Arr[8] := FALSE;
   S711AB_KEY_CARTYPE.STN_Btype_6Arr[9] := FALSE;
   S711AB_KEY_CARTYPE.STN_Btype_6Arr[10] := FALSE;
   S711AB_KEY_CARTYPE.STN_Btype_6Arr[11] := FALSE;
   S711AB_KEY_CARTYPE.STN_Btype_6Arr[12] := FALSE;
   S711AB_KEY_CARTYPE.STN_Btype_6Arr[13] := FALSE;
   S711AB_KEY_CARTYPE.STN_Btype_6Arr[14] := FALSE;
   S711AB_KEY_CARTYPE.STN_Btype_6Arr[15] := FALSE;
   S711AB_KEY_CARTYPE.STN_1st_BT_On := FALSE;
   S711AB_KEY_CARTYPE.STN_2nd_BT_On := FALSE;
   S711AB_KEY_CARTYPE.STN_3rd_BT_On := FALSE;
   S711AB_KEY_CARTYPE.STN_4th_BT_On := FALSE;
   S711AB_KEY_CARTYPE.STN_5th_BT_On := FALSE;
   S711AB_KEY_CARTYPE.STN_6th_BT_On := FALSE;
   S711AB_KEY_CARTYPE.STN_7th_BT_On := FALSE;
   S711AB_KEY_CARTYPE.STN_8th_BT_On := FALSE;
   S711AB_KEY_CARTYPE.STN_9th_BT_On := FALSE;
   S711AB_KEY_CARTYPE.STN_10th_BT_On := FALSE;
   S711AB_KEY_CARTYPE.STN_11th_BT_On := FALSE;
   S711AB_KEY_CARTYPE.STN_12th_BT_On := FALSE;
   S711AB_KEY_CARTYPE.STN_1st_BT_Off := FALSE;
   S711AB_KEY_CARTYPE.BLKMove_Ret := 0;
   S711AB_KEY_CARTYPE.VIN_1BCD := W#16#0;
   S711AB_KEY_CARTYPE.VIN_2BCD := W#16#0;
   S711AB_KEY_CARTYPE.VIN_1Int := 0;
   S711AB_KEY_CARTYPE.VIN_2Int := 0;
   S711A_R1_CARTYPE.Stn_Vin_No := L#0;
   S711A_R1_CARTYPE.Stn_Bt_1Word := W#16#0;
   S711A_R1_CARTYPE.Stn_Bt_2Word := W#16#0;
   S711A_R1_CARTYPE.Stn_Bt_3Word := W#16#0;
   S711A_R1_CARTYPE.Stn_Bt_4Word := W#16#0;
   S711A_R1_CARTYPE.Stn_Bt_5Word_Sp := W#16#0;
   S711A_R1_CARTYPE.Stn_Bt_6Word_Sp := W#16#0;
   S711A_R1_CARTYPE.M_BType_On := FALSE;
   S711A_R1_CARTYPE.M_BType_None := FALSE;
   S711A_R1_CARTYPE.M_Bypass_BType := FALSE;
   S711A_R1_CARTYPE.M_BType_TL := FALSE;
   S711A_R1_CARTYPE.M_BType_LM := FALSE;
   S711A_R1_CARTYPE.M_BType_SP1 := FALSE;
   S711A_R1_CARTYPE.M_BType_SP2 := FALSE;
   S711A_R1_CARTYPE.M_BType_SP3 := FALSE;
   S711A_R1_CARTYPE.M_BType_DOM := FALSE;
   S711A_R1_CARTYPE.M_BType_EXP := FALSE;
   S711A_R1_CARTYPE.Robot_Prog_No := 0;
   S711A_R1_CARTYPE.STN_Btype_1Arr[0] := FALSE;
   S711A_R1_CARTYPE.STN_Btype_1Arr[1] := FALSE;
   S711A_R1_CARTYPE.STN_Btype_1Arr[2] := FALSE;
   S711A_R1_CARTYPE.STN_Btype_1Arr[3] := FALSE;
   S711A_R1_CARTYPE.STN_Btype_1Arr[4] := FALSE;
   S711A_R1_CARTYPE.STN_Btype_1Arr[5] := FALSE;
   S711A_R1_CARTYPE.STN_Btype_1Arr[6] := FALSE;
   S711A_R1_CARTYPE.STN_Btype_1Arr[7] := FALSE;
   S711A_R1_CARTYPE.STN_Btype_1Arr[8] := FALSE;
   S711A_R1_CARTYPE.STN_Btype_1Arr[9] := FALSE;
   S711A_R1_CARTYPE.STN_Btype_1Arr[10] := FALSE;
   S711A_R1_CARTYPE.STN_Btype_1Arr[11] := FALSE;
   S711A_R1_CARTYPE.STN_Btype_1Arr[12] := FALSE;
   S711A_R1_CARTYPE.STN_Btype_1Arr[13] := FALSE;
   S711A_R1_CARTYPE.STN_Btype_1Arr[14] := FALSE;
   S711A_R1_CARTYPE.STN_Btype_1Arr[15] := FALSE;
   S711A_R1_CARTYPE.STN_Btype_2Arr[0] := FALSE;
   S711A_R1_CARTYPE.STN_Btype_2Arr[1] := FALSE;
   S711A_R1_CARTYPE.STN_Btype_2Arr[2] := FALSE;
   S711A_R1_CARTYPE.STN_Btype_2Arr[3] := FALSE;
   S711A_R1_CARTYPE.STN_Btype_2Arr[4] := FALSE;
   S711A_R1_CARTYPE.STN_Btype_2Arr[5] := FALSE;
   S711A_R1_CARTYPE.STN_Btype_2Arr[6] := FALSE;
   S711A_R1_CARTYPE.STN_Btype_2Arr[7] := FALSE;
   S711A_R1_CARTYPE.STN_Btype_2Arr[8] := FALSE;
   S711A_R1_CARTYPE.STN_Btype_2Arr[9] := FALSE;
   S711A_R1_CARTYPE.STN_Btype_2Arr[10] := FALSE;
   S711A_R1_CARTYPE.STN_Btype_2Arr[11] := FALSE;
   S711A_R1_CARTYPE.STN_Btype_2Arr[12] := FALSE;
   S711A_R1_CARTYPE.STN_Btype_2Arr[13] := FALSE;
   S711A_R1_CARTYPE.STN_Btype_2Arr[14] := FALSE;
   S711A_R1_CARTYPE.STN_Btype_2Arr[15] := FALSE;
   S711A_R1_CARTYPE.STN_Btype_3Arr[0] := FALSE;
   S711A_R1_CARTYPE.STN_Btype_3Arr[1] := FALSE;
   S711A_R1_CARTYPE.STN_Btype_3Arr[2] := FALSE;
   S711A_R1_CARTYPE.STN_Btype_3Arr[3] := FALSE;
   S711A_R1_CARTYPE.STN_Btype_3Arr[4] := FALSE;
   S711A_R1_CARTYPE.STN_Btype_3Arr[5] := FALSE;
   S711A_R1_CARTYPE.STN_Btype_3Arr[6] := FALSE;
   S711A_R1_CARTYPE.STN_Btype_3Arr[7] := FALSE;
   S711A_R1_CARTYPE.STN_Btype_3Arr[8] := FALSE;
   S711A_R1_CARTYPE.STN_Btype_3Arr[9] := FALSE;
   S711A_R1_CARTYPE.STN_Btype_3Arr[10] := FALSE;
   S711A_R1_CARTYPE.STN_Btype_3Arr[11] := FALSE;
   S711A_R1_CARTYPE.STN_Btype_3Arr[12] := FALSE;
   S711A_R1_CARTYPE.STN_Btype_3Arr[13] := FALSE;
   S711A_R1_CARTYPE.STN_Btype_3Arr[14] := FALSE;
   S711A_R1_CARTYPE.STN_Btype_3Arr[15] := FALSE;
   S711A_R1_CARTYPE.STN_Btype_4Arr[0] := FALSE;
   S711A_R1_CARTYPE.STN_Btype_4Arr[1] := FALSE;
   S711A_R1_CARTYPE.STN_Btype_4Arr[2] := FALSE;
   S711A_R1_CARTYPE.STN_Btype_4Arr[3] := FALSE;
   S711A_R1_CARTYPE.STN_Btype_4Arr[4] := FALSE;
   S711A_R1_CARTYPE.STN_Btype_4Arr[5] := FALSE;
   S711A_R1_CARTYPE.STN_Btype_4Arr[6] := FALSE;
   S711A_R1_CARTYPE.STN_Btype_4Arr[7] := FALSE;
   S711A_R1_CARTYPE.STN_Btype_4Arr[8] := FALSE;
   S711A_R1_CARTYPE.STN_Btype_4Arr[9] := FALSE;
   S711A_R1_CARTYPE.STN_Btype_4Arr[10] := FALSE;
   S711A_R1_CARTYPE.STN_Btype_4Arr[11] := FALSE;
   S711A_R1_CARTYPE.STN_Btype_4Arr[12] := FALSE;
   S711A_R1_CARTYPE.STN_Btype_4Arr[13] := FALSE;
   S711A_R1_CARTYPE.STN_Btype_4Arr[14] := FALSE;
   S711A_R1_CARTYPE.STN_Btype_4Arr[15] := FALSE;
   S711A_R1_CARTYPE.STN_Btype_5Arr[0] := FALSE;
   S711A_R1_CARTYPE.STN_Btype_5Arr[1] := FALSE;
   S711A_R1_CARTYPE.STN_Btype_5Arr[2] := FALSE;
   S711A_R1_CARTYPE.STN_Btype_5Arr[3] := FALSE;
   S711A_R1_CARTYPE.STN_Btype_5Arr[4] := FALSE;
   S711A_R1_CARTYPE.STN_Btype_5Arr[5] := FALSE;
   S711A_R1_CARTYPE.STN_Btype_5Arr[6] := FALSE;
   S711A_R1_CARTYPE.STN_Btype_5Arr[7] := FALSE;
   S711A_R1_CARTYPE.STN_Btype_5Arr[8] := FALSE;
   S711A_R1_CARTYPE.STN_Btype_5Arr[9] := FALSE;
   S711A_R1_CARTYPE.STN_Btype_5Arr[10] := FALSE;
   S711A_R1_CARTYPE.STN_Btype_5Arr[11] := FALSE;
   S711A_R1_CARTYPE.STN_Btype_5Arr[12] := FALSE;
   S711A_R1_CARTYPE.STN_Btype_5Arr[13] := FALSE;
   S711A_R1_CARTYPE.STN_Btype_5Arr[14] := FALSE;
   S711A_R1_CARTYPE.STN_Btype_5Arr[15] := FALSE;
   S711A_R1_CARTYPE.STN_Btype_6Arr[0] := FALSE;
   S711A_R1_CARTYPE.STN_Btype_6Arr[1] := FALSE;
   S711A_R1_CARTYPE.STN_Btype_6Arr[2] := FALSE;
   S711A_R1_CARTYPE.STN_Btype_6Arr[3] := FALSE;
   S711A_R1_CARTYPE.STN_Btype_6Arr[4] := FALSE;
   S711A_R1_CARTYPE.STN_Btype_6Arr[5] := FALSE;
   S711A_R1_CARTYPE.STN_Btype_6Arr[6] := FALSE;
   S711A_R1_CARTYPE.STN_Btype_6Arr[7] := FALSE;
   S711A_R1_CARTYPE.STN_Btype_6Arr[8] := FALSE;
   S711A_R1_CARTYPE.STN_Btype_6Arr[9] := FALSE;
   S711A_R1_CARTYPE.STN_Btype_6Arr[10] := FALSE;
   S711A_R1_CARTYPE.STN_Btype_6Arr[11] := FALSE;
   S711A_R1_CARTYPE.STN_Btype_6Arr[12] := FALSE;
   S711A_R1_CARTYPE.STN_Btype_6Arr[13] := FALSE;
   S711A_R1_CARTYPE.STN_Btype_6Arr[14] := FALSE;
   S711A_R1_CARTYPE.STN_Btype_6Arr[15] := FALSE;
   S711A_R1_CARTYPE.STN_1st_BT_On := FALSE;
   S711A_R1_CARTYPE.STN_2nd_BT_On := FALSE;
   S711A_R1_CARTYPE.STN_3rd_BT_On := FALSE;
   S711A_R1_CARTYPE.STN_4th_BT_On := FALSE;
   S711A_R1_CARTYPE.STN_5th_BT_On := FALSE;
   S711A_R1_CARTYPE.STN_6th_BT_On := FALSE;
   S711A_R1_CARTYPE.STN_7th_BT_On := FALSE;
   S711A_R1_CARTYPE.STN_8th_BT_On := FALSE;
   S711A_R1_CARTYPE.STN_9th_BT_On := FALSE;
   S711A_R1_CARTYPE.STN_10th_BT_On := FALSE;
   S711A_R1_CARTYPE.STN_11th_BT_On := FALSE;
   S711A_R1_CARTYPE.STN_12th_BT_On := FALSE;
   S711A_R1_CARTYPE.STN_1st_BT_Off := FALSE;
   S711A_R1_CARTYPE.BLKMove_Ret := 0;
   S711A_R1_CARTYPE.VIN_1BCD := W#16#0;
   S711A_R1_CARTYPE.VIN_2BCD := W#16#0;
   S711A_R1_CARTYPE.VIN_1Int := 0;
   S711A_R1_CARTYPE.VIN_2Int := 0;
   S711_IDLE_CARTYPE.Stn_Vin_No := L#0;
   S711_IDLE_CARTYPE.Stn_Bt_1Word := W#16#0;
   S711_IDLE_CARTYPE.Stn_Bt_2Word := W#16#0;
   S711_IDLE_CARTYPE.Stn_Bt_3Word := W#16#0;
   S711_IDLE_CARTYPE.Stn_Bt_4Word := W#16#0;
   S711_IDLE_CARTYPE.Stn_Bt_5Word_Sp := W#16#0;
   S711_IDLE_CARTYPE.Stn_Bt_6Word_Sp := W#16#0;
   S711_IDLE_CARTYPE.M_BType_On := FALSE;
   S711_IDLE_CARTYPE.M_BType_None := FALSE;
   S711_IDLE_CARTYPE.M_Bypass_BType := FALSE;
   S711_IDLE_CARTYPE.M_BType_TL := FALSE;
   S711_IDLE_CARTYPE.M_BType_LM := FALSE;
   S711_IDLE_CARTYPE.M_BType_SP1 := FALSE;
   S711_IDLE_CARTYPE.M_BType_SP2 := FALSE;
   S711_IDLE_CARTYPE.M_BType_SP3 := FALSE;
   S711_IDLE_CARTYPE.M_BType_DOM := FALSE;
   S711_IDLE_CARTYPE.M_BType_EXP := FALSE;
   S711_IDLE_CARTYPE.Robot_Prog_No := 0;
   S711_IDLE_CARTYPE.STN_Btype_1Arr[0] := FALSE;
   S711_IDLE_CARTYPE.STN_Btype_1Arr[1] := FALSE;
   S711_IDLE_CARTYPE.STN_Btype_1Arr[2] := FALSE;
   S711_IDLE_CARTYPE.STN_Btype_1Arr[3] := FALSE;
   S711_IDLE_CARTYPE.STN_Btype_1Arr[4] := FALSE;
   S711_IDLE_CARTYPE.STN_Btype_1Arr[5] := FALSE;
   S711_IDLE_CARTYPE.STN_Btype_1Arr[6] := FALSE;
   S711_IDLE_CARTYPE.STN_Btype_1Arr[7] := FALSE;
   S711_IDLE_CARTYPE.STN_Btype_1Arr[8] := FALSE;
   S711_IDLE_CARTYPE.STN_Btype_1Arr[9] := FALSE;
   S711_IDLE_CARTYPE.STN_Btype_1Arr[10] := FALSE;
   S711_IDLE_CARTYPE.STN_Btype_1Arr[11] := FALSE;
   S711_IDLE_CARTYPE.STN_Btype_1Arr[12] := FALSE;
   S711_IDLE_CARTYPE.STN_Btype_1Arr[13] := FALSE;
   S711_IDLE_CARTYPE.STN_Btype_1Arr[14] := FALSE;
   S711_IDLE_CARTYPE.STN_Btype_1Arr[15] := FALSE;
   S711_IDLE_CARTYPE.STN_Btype_2Arr[0] := FALSE;
   S711_IDLE_CARTYPE.STN_Btype_2Arr[1] := FALSE;
   S711_IDLE_CARTYPE.STN_Btype_2Arr[2] := FALSE;
   S711_IDLE_CARTYPE.STN_Btype_2Arr[3] := FALSE;
   S711_IDLE_CARTYPE.STN_Btype_2Arr[4] := FALSE;
   S711_IDLE_CARTYPE.STN_Btype_2Arr[5] := FALSE;
   S711_IDLE_CARTYPE.STN_Btype_2Arr[6] := FALSE;
   S711_IDLE_CARTYPE.STN_Btype_2Arr[7] := FALSE;
   S711_IDLE_CARTYPE.STN_Btype_2Arr[8] := FALSE;
   S711_IDLE_CARTYPE.STN_Btype_2Arr[9] := FALSE;
   S711_IDLE_CARTYPE.STN_Btype_2Arr[10] := FALSE;
   S711_IDLE_CARTYPE.STN_Btype_2Arr[11] := FALSE;
   S711_IDLE_CARTYPE.STN_Btype_2Arr[12] := FALSE;
   S711_IDLE_CARTYPE.STN_Btype_2Arr[13] := FALSE;
   S711_IDLE_CARTYPE.STN_Btype_2Arr[14] := FALSE;
   S711_IDLE_CARTYPE.STN_Btype_2Arr[15] := FALSE;
   S711_IDLE_CARTYPE.STN_Btype_3Arr[0] := FALSE;
   S711_IDLE_CARTYPE.STN_Btype_3Arr[1] := FALSE;
   S711_IDLE_CARTYPE.STN_Btype_3Arr[2] := FALSE;
   S711_IDLE_CARTYPE.STN_Btype_3Arr[3] := FALSE;
   S711_IDLE_CARTYPE.STN_Btype_3Arr[4] := FALSE;
   S711_IDLE_CARTYPE.STN_Btype_3Arr[5] := FALSE;
   S711_IDLE_CARTYPE.STN_Btype_3Arr[6] := FALSE;
   S711_IDLE_CARTYPE.STN_Btype_3Arr[7] := FALSE;
   S711_IDLE_CARTYPE.STN_Btype_3Arr[8] := FALSE;
   S711_IDLE_CARTYPE.STN_Btype_3Arr[9] := FALSE;
   S711_IDLE_CARTYPE.STN_Btype_3Arr[10] := FALSE;
   S711_IDLE_CARTYPE.STN_Btype_3Arr[11] := FALSE;
   S711_IDLE_CARTYPE.STN_Btype_3Arr[12] := FALSE;
   S711_IDLE_CARTYPE.STN_Btype_3Arr[13] := FALSE;
   S711_IDLE_CARTYPE.STN_Btype_3Arr[14] := FALSE;
   S711_IDLE_CARTYPE.STN_Btype_3Arr[15] := FALSE;
   S711_IDLE_CARTYPE.STN_Btype_4Arr[0] := FALSE;
   S711_IDLE_CARTYPE.STN_Btype_4Arr[1] := FALSE;
   S711_IDLE_CARTYPE.STN_Btype_4Arr[2] := FALSE;
   S711_IDLE_CARTYPE.STN_Btype_4Arr[3] := FALSE;
   S711_IDLE_CARTYPE.STN_Btype_4Arr[4] := FALSE;
   S711_IDLE_CARTYPE.STN_Btype_4Arr[5] := FALSE;
   S711_IDLE_CARTYPE.STN_Btype_4Arr[6] := FALSE;
   S711_IDLE_CARTYPE.STN_Btype_4Arr[7] := FALSE;
   S711_IDLE_CARTYPE.STN_Btype_4Arr[8] := FALSE;
   S711_IDLE_CARTYPE.STN_Btype_4Arr[9] := FALSE;
   S711_IDLE_CARTYPE.STN_Btype_4Arr[10] := FALSE;
   S711_IDLE_CARTYPE.STN_Btype_4Arr[11] := FALSE;
   S711_IDLE_CARTYPE.STN_Btype_4Arr[12] := FALSE;
   S711_IDLE_CARTYPE.STN_Btype_4Arr[13] := FALSE;
   S711_IDLE_CARTYPE.STN_Btype_4Arr[14] := FALSE;
   S711_IDLE_CARTYPE.STN_Btype_4Arr[15] := FALSE;
   S711_IDLE_CARTYPE.STN_Btype_5Arr[0] := FALSE;
   S711_IDLE_CARTYPE.STN_Btype_5Arr[1] := FALSE;
   S711_IDLE_CARTYPE.STN_Btype_5Arr[2] := FALSE;
   S711_IDLE_CARTYPE.STN_Btype_5Arr[3] := FALSE;
   S711_IDLE_CARTYPE.STN_Btype_5Arr[4] := FALSE;
   S711_IDLE_CARTYPE.STN_Btype_5Arr[5] := FALSE;
   S711_IDLE_CARTYPE.STN_Btype_5Arr[6] := FALSE;
   S711_IDLE_CARTYPE.STN_Btype_5Arr[7] := FALSE;
   S711_IDLE_CARTYPE.STN_Btype_5Arr[8] := FALSE;
   S711_IDLE_CARTYPE.STN_Btype_5Arr[9] := FALSE;
   S711_IDLE_CARTYPE.STN_Btype_5Arr[10] := FALSE;
   S711_IDLE_CARTYPE.STN_Btype_5Arr[11] := FALSE;
   S711_IDLE_CARTYPE.STN_Btype_5Arr[12] := FALSE;
   S711_IDLE_CARTYPE.STN_Btype_5Arr[13] := FALSE;
   S711_IDLE_CARTYPE.STN_Btype_5Arr[14] := FALSE;
   S711_IDLE_CARTYPE.STN_Btype_5Arr[15] := FALSE;
   S711_IDLE_CARTYPE.STN_Btype_6Arr[0] := FALSE;
   S711_IDLE_CARTYPE.STN_Btype_6Arr[1] := FALSE;
   S711_IDLE_CARTYPE.STN_Btype_6Arr[2] := FALSE;
   S711_IDLE_CARTYPE.STN_Btype_6Arr[3] := FALSE;
   S711_IDLE_CARTYPE.STN_Btype_6Arr[4] := FALSE;
   S711_IDLE_CARTYPE.STN_Btype_6Arr[5] := FALSE;
   S711_IDLE_CARTYPE.STN_Btype_6Arr[6] := FALSE;
   S711_IDLE_CARTYPE.STN_Btype_6Arr[7] := FALSE;
   S711_IDLE_CARTYPE.STN_Btype_6Arr[8] := FALSE;
   S711_IDLE_CARTYPE.STN_Btype_6Arr[9] := FALSE;
   S711_IDLE_CARTYPE.STN_Btype_6Arr[10] := FALSE;
   S711_IDLE_CARTYPE.STN_Btype_6Arr[11] := FALSE;
   S711_IDLE_CARTYPE.STN_Btype_6Arr[12] := FALSE;
   S711_IDLE_CARTYPE.STN_Btype_6Arr[13] := FALSE;
   S711_IDLE_CARTYPE.STN_Btype_6Arr[14] := FALSE;
   S711_IDLE_CARTYPE.STN_Btype_6Arr[15] := FALSE;
   S711_IDLE_CARTYPE.STN_1st_BT_On := FALSE;
   S711_IDLE_CARTYPE.STN_2nd_BT_On := FALSE;
   S711_IDLE_CARTYPE.STN_3rd_BT_On := FALSE;
   S711_IDLE_CARTYPE.STN_4th_BT_On := FALSE;
   S711_IDLE_CARTYPE.STN_5th_BT_On := FALSE;
   S711_IDLE_CARTYPE.STN_6th_BT_On := FALSE;
   S711_IDLE_CARTYPE.STN_7th_BT_On := FALSE;
   S711_IDLE_CARTYPE.STN_8th_BT_On := FALSE;
   S711_IDLE_CARTYPE.STN_9th_BT_On := FALSE;
   S711_IDLE_CARTYPE.STN_10th_BT_On := FALSE;
   S711_IDLE_CARTYPE.STN_11th_BT_On := FALSE;
   S711_IDLE_CARTYPE.STN_12th_BT_On := FALSE;
   S711_IDLE_CARTYPE.STN_1st_BT_Off := FALSE;
   S711_IDLE_CARTYPE.BLKMove_Ret := 0;
   S711_IDLE_CARTYPE.VIN_1BCD := W#16#0;
   S711_IDLE_CARTYPE.VIN_2BCD := W#16#0;
   S711_IDLE_CARTYPE.VIN_1Int := 0;
   S711_IDLE_CARTYPE.VIN_2Int := 0;
END_DATA_BLOCK

FUNCTION FC 106 : VOID
TITLE =BODY TYPE PROGRAM
VERSION : 0.1

BEGIN
NETWORK
TITLE =ONLY ZERO
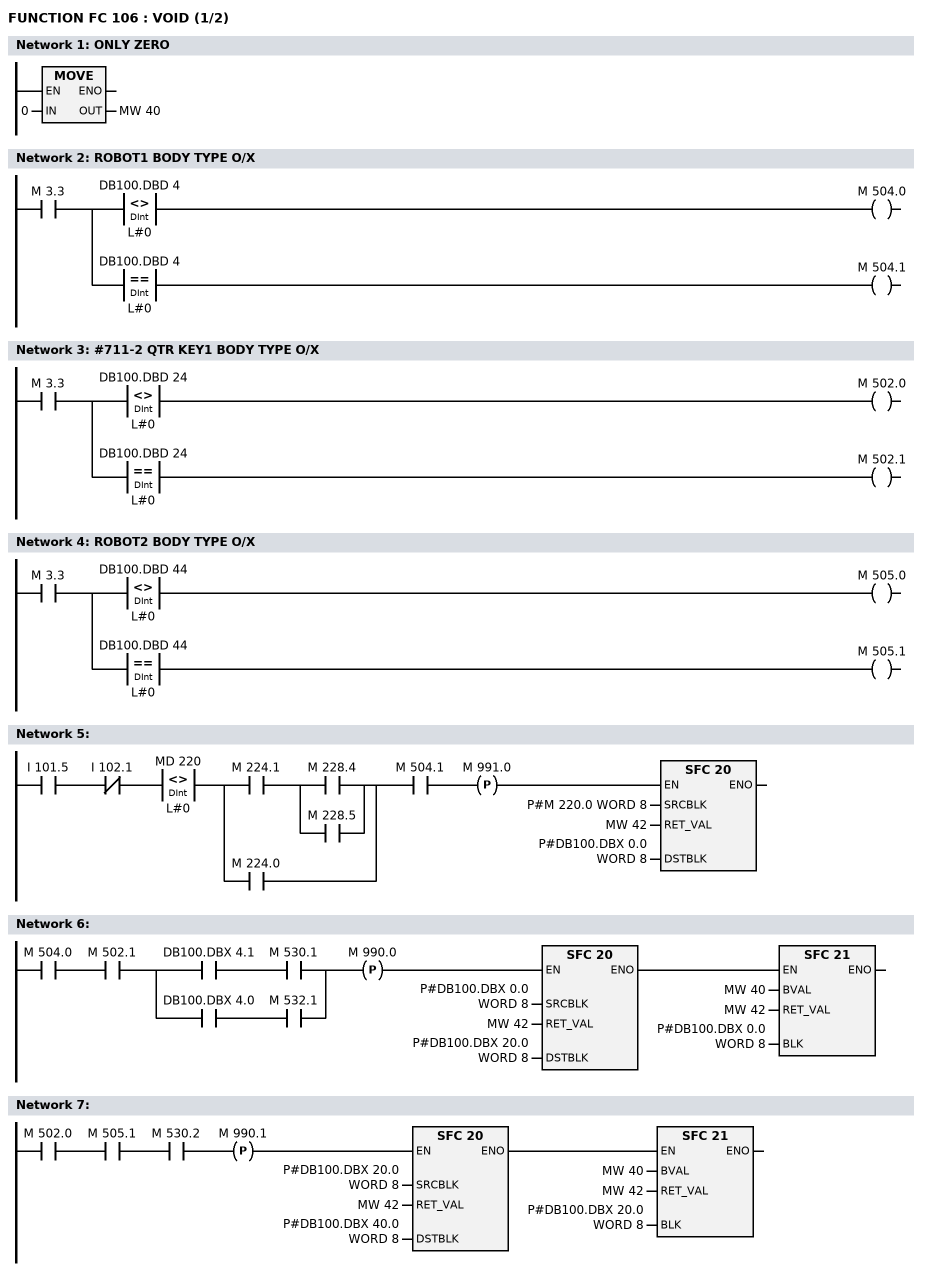

      L     0;
      T     MW    40;
      NOP   0;
NETWORK
TITLE =ROBOT1 BODY TYPE O/X

      A     M      3.3;
      =     L      0.0;
      A     L      0.0;
      A(    ;
      L     DB100.DBD    4;
      L     L#0;
      <>D   ;
      )     ;
      =     M    504.0;
      A     L      0.0;
      A(    ;
      L     DB100.DBD    4;
      L     L#0;
      ==D   ;
      )     ;
      =     M    504.1;
NETWORK
TITLE =#711-2 QTR KEY1 BODY TYPE O/X

      A     M      3.3;
      =     L      0.0;
      A     L      0.0;
      A(    ;
      L     DB100.DBD   24;
      L     L#0;
      <>D   ;
      )     ;
      =     M    502.0;
      A     L      0.0;
      A(    ;
      L     DB100.DBD   24;
      L     L#0;
      ==D   ;
      )     ;
      =     M    502.1;
NETWORK
TITLE =ROBOT2 BODY TYPE O/X

      A     M      3.3;
      =     L      0.0;
      A     L      0.0;
      A(    ;
      L     DB100.DBD   44;
      L     L#0;
      <>D   ;
      )     ;
      =     M    505.0;
      A     L      0.0;
      A(    ;
      L     DB100.DBD   44;
      L     L#0;
      ==D   ;
      )     ;
      =     M    505.1;
NETWORK
TITLE =

      A     I    101.5;
      AN    I    102.1;
      A(    ;
      L     MD   220;
      L     L#0;
      <>D   ;
      )     ;
      A(    ;
      A     M    224.1;
      A(    ;
      O     M    228.4;
      O     M    228.5;
      )     ;
      O     M    224.0;
      )     ;
      A     M    504.1;
      FP    M    991.0;
      JNB   _001;
      CALL SFC   20 (
           SRCBLK                   := P#M 220.0 WORD 8,
           RET_VAL                  := MW    42,
           DSTBLK                   := P#DB100.DBX 0.0 WORD 8);
_001: NOP   0;
NETWORK
TITLE =

      A(    ;
      A     M    504.0;
      A     M    502.1;
      A(    ;
      A     DB100.DBX    4.1;
      A     M    530.1;
      O     ;
      A     DB100.DBX    4.0;
      A     M    532.1;
      )     ;
      FP    M    990.0;
      JNB   _002;
      CALL SFC   20 (
           SRCBLK                   := P#DB100.DBX 0.0 WORD 8,
           RET_VAL                  := MW    42,
           DSTBLK                   := P#DB100.DBX 20.0 WORD 8);
_002: A     BR;
      )     ;
      JNB   _003;
      CALL SFC   21 (
           BVAL                     := MW    40,
           RET_VAL                  := MW    42,
           BLK                      := P#DB100.DBX 0.0 WORD 8);
_003: NOP   0;
NETWORK
TITLE =

      A(    ;
      A     M    502.0;
      A     M    505.1;
      A     M    530.2;
      FP    M    990.1;
      JNB   _004;
      CALL SFC   20 (
           SRCBLK                   := P#DB100.DBX 20.0 WORD 8,
           RET_VAL                  := MW    42,
           DSTBLK                   := P#DB100.DBX 40.0 WORD 8);
_004: A     BR;
      )     ;
      JNB   _005;
      CALL SFC   21 (
           BVAL                     := MW    40,
           RET_VAL                  := MW    42,
           BLK                      := P#DB100.DBX 20.0 WORD 8);
_005: NOP   0;
NETWORK
TITLE =
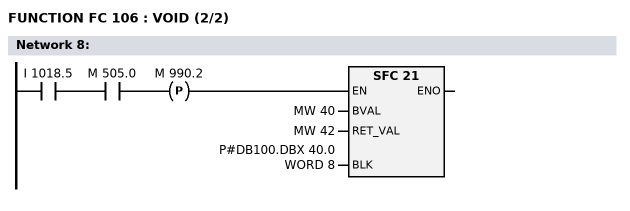

      A     I   1018.5;
      A     M    505.0;
      FP    M    990.2;
      JNB   _006;
      CALL SFC   21 (
           BVAL                     := MW    40,
           RET_VAL                  := MW    42,
           BLK                      := P#DB100.DBX 40.0 WORD 8);
_006: NOP   0;
END_FUNCTION

FUNCTION_BLOCK FB 108
TITLE =
VERSION : 0.1

BEGIN
NETWORK
TITLE =PROFINET ERROR(1~10)
//
//
      A     M      3.3;
      =     L      0.0;
      A     L      0.0;
      A(    ;
      O     DB327.DBX 1025.3;
      O     ;
      A     M   7000.0;
      AN    I    100.1;
      AN    I      0.1;
      )     ;
      =     L      0.1;
      A     L      0.1;
      A     T    700;
      =     M   7000.0;
      A     L      0.1;
      BLD   102;
      L     S5T#0MS;
      SD    T    700;
      A     L      0.0;
      A(    ;
      O     DB327.DBX 1027.3;
      O     ;
      A     M   7000.1;
      AN    I    100.1;
      AN    I      0.1;
      )     ;
      =     L      0.1;
      A     L      0.1;
      A     T    701;
      =     M   7000.1;
      A     L      0.1;
      BLD   102;
      L     S5T#0MS;
      SD    T    701;
      A     L      0.0;
      A(    ;
      O     DB327.DBX 1029.3;
      O     ;
      A     M   7000.2;
      AN    I    100.1;
      AN    I      0.1;
      )     ;
      =     L      0.1;
      A     L      0.1;
      A     T    702;
      =     M   7000.2;
      A     L      0.1;
      BLD   102;
      L     S5T#0MS;
      SD    T    702;
      A     L      0.0;
      A(    ;
      O     DB327.DBX 1031.3;
      O     ;
      A     M   7000.3;
      AN    I    100.1;
      AN    I      0.1;
      )     ;
      =     L      0.1;
      A     L      0.1;
      A     T    703;
      =     M   7000.3;
      A     L      0.1;
      BLD   102;
      L     S5T#0MS;
      SD    T    703;
      A     L      0.0;
      A(    ;
      O     DB327.DBX 1033.3;
      O     ;
      A     M   7000.4;
      AN    I    100.1;
      AN    I      0.1;
      )     ;
      =     L      0.1;
      A     L      0.1;
      A     T    704;
      =     M   7000.4;
      A     L      0.1;
      BLD   102;
      L     S5T#0MS;
      SD    T    704;
      A     L      0.0;
      A(    ;
      O     DB327.DBX 1035.3;
      O     ;
      A     M   7000.5;
      AN    I    100.1;
      AN    I      0.1;
      )     ;
      =     L      0.1;
      A     L      0.1;
      A     T    705;
      =     M   7000.5;
      A     L      0.1;
      BLD   102;
      L     S5T#0MS;
      SD    T    705;
      A     L      0.0;
      A(    ;
      O     DB327.DBX 1037.3;
      O     ;
      A     M   7000.6;
      AN    I    100.1;
      AN    I      0.1;
      )     ;
      =     L      0.1;
      A     L      0.1;
      A     T    706;
      =     M   7000.6;
      A     L      0.1;
      BLD   102;
      L     S5T#0MS;
      SD    T    706;
      A     L      0.0;
      A(    ;
      O     DB327.DBX 1039.3;
      O     ;
      A     M   7000.7;
      AN    I    100.1;
      AN    I      0.1;
      )     ;
      =     L      0.1;
      A     L      0.1;
      A     T    707;
      =     M   7000.7;
      A     L      0.1;
      BLD   102;
      L     S5T#0MS;
      SD    T    707;
      A     L      0.0;
      A(    ;
      O     DB327.DBX 1041.3;
      O     ;
      A     M   7001.0;
      AN    I    100.1;
      AN    I      0.1;
      )     ;
      =     L      0.1;
      A     L      0.1;
      A     T    708;
      =     M   7001.0;
      A     L      0.1;
      BLD   102;
      L     S5T#0MS;
      SD    T    708;
      A     L      0.0;
      A(    ;
      O     DB327.DBX 1043.3;
      O     ;
      A     M   7001.1;
      AN    I    100.1;
      AN    I      0.1;
      )     ;
      =     L      0.1;
      A     L      0.1;
      A     T    709;
      =     M   7001.1;
      A     L      0.1;
      BLD   102;
      L     S5T#0MS;
      SD    T    709;
NETWORK
TITLE =PROFINET ERROR(11~20)
//
//
      A     M      3.3;
      =     L      0.0;
      A     L      0.0;
      A(    ;
      O     DB327.DBX 1045.3;
      O     ;
      A     M   7001.2;
      AN    I    100.1;
      AN    I      0.1;
      )     ;
      =     L      0.1;
      A     L      0.1;
      A     T    710;
      =     M   7001.2;
      A     L      0.1;
      BLD   102;
      L     S5T#0MS;
      SD    T    710;
      A     L      0.0;
      A(    ;
      O     DB327.DBX 1047.3;
      O     ;
      A     M   7001.3;
      AN    I    100.1;
      AN    I      0.1;
      )     ;
      =     L      0.1;
      A     L      0.1;
      A     T    711;
      =     M   7001.3;
      A     L      0.1;
      BLD   102;
      L     S5T#0MS;
      SD    T    711;
      A     L      0.0;
      A(    ;
      O     DB327.DBX 1049.3;
      O     ;
      A     M   7001.4;
      AN    I    100.1;
      AN    I      0.1;
      )     ;
      =     L      0.1;
      A     L      0.1;
      A     T    712;
      =     M   7001.4;
      A     L      0.1;
      BLD   102;
      L     S5T#0MS;
      SD    T    712;
      A     L      0.0;
      A(    ;
      O     DB327.DBX 1051.3;
      O     ;
      A     M   7001.5;
      AN    I    100.1;
      AN    I      0.1;
      )     ;
      =     L      0.1;
      A     L      0.1;
      A     T    713;
      =     M   7001.5;
      A     L      0.1;
      BLD   102;
      L     S5T#0MS;
      SD    T    713;
      A     L      0.0;
      A(    ;
      O     DB327.DBX 1053.3;
      O     ;
      A     M   7001.6;
      AN    I    100.1;
      AN    I      0.1;
      )     ;
      =     L      0.1;
      A     L      0.1;
      A     T    714;
      =     M   7001.6;
      A     L      0.1;
      BLD   102;
      L     S5T#0MS;
      SD    T    714;
      A     L      0.0;
      A(    ;
      O     DB327.DBX 1055.3;
      O     ;
      A     M   7001.7;
      AN    I    100.1;
      AN    I      0.1;
      )     ;
      =     L      0.1;
      A     L      0.1;
      A     T    715;
      =     M   7001.7;
      A     L      0.1;
      BLD   102;
      L     S5T#0MS;
      SD    T    715;
      A     L      0.0;
      A(    ;
      O     DB327.DBX 1057.3;
      O     ;
      A     M   7002.0;
      AN    I    100.1;
      AN    I      0.1;
      )     ;
      =     L      0.1;
      A     L      0.1;
      A     T    716;
      =     M   7002.0;
      A     L      0.1;
      BLD   102;
      L     S5T#0MS;
      SD    T    716;
      A     L      0.0;
      A(    ;
      O     DB327.DBX 1059.3;
      O     ;
      A     M   7002.1;
      AN    I    100.1;
      AN    I      0.1;
      )     ;
      =     L      0.1;
      A     L      0.1;
      A     T    717;
      =     M   7002.1;
      A     L      0.1;
      BLD   102;
      L     S5T#0MS;
      SD    T    717;
      A     L      0.0;
      A(    ;
      O     DB327.DBX 1061.3;
      O     ;
      A     M   7002.2;
      AN    I    100.1;
      AN    I      0.1;
      )     ;
      =     L      0.1;
      A     L      0.1;
      A     T    718;
      =     M   7002.2;
      A     L      0.1;
      BLD   102;
      L     S5T#0MS;
      SD    T    718;
      A     L      0.0;
      A(    ;
      O     DB327.DBX 1063.3;
      O     ;
      A     M   7002.3;
      AN    I    100.1;
      AN    I      0.1;
      )     ;
      =     L      0.1;
      A     L      0.1;
      A     T    719;
      =     M   7002.3;
      A     L      0.1;
      BLD   102;
      L     S5T#0MS;
      SD    T    719;
NETWORK
TITLE =PROFINET ERROR(21~30)
//
//
      A     M      3.3;
      =     L      0.0;
      A     L      0.0;
      A(    ;
      O     DB327.DBX 1065.3;
      O     ;
      A     M   7002.4;
      AN    I    100.1;
      AN    I      0.1;
      )     ;
      =     L      0.1;
      A     L      0.1;
      A     T    720;
      =     M   7002.4;
      A     L      0.1;
      BLD   102;
      L     S5T#0MS;
      SD    T    720;
      A     L      0.0;
      A(    ;
      O     DB327.DBX 1067.3;
      O     ;
      A     M   7002.5;
      AN    I    100.1;
      AN    I      0.1;
      )     ;
      =     L      0.1;
      A     L      0.1;
      A     T    721;
      =     M   7002.5;
      A     L      0.1;
      BLD   102;
      L     S5T#0MS;
      SD    T    721;
      A     L      0.0;
      A(    ;
      O     DB327.DBX 1069.3;
      O     ;
      A     M   7002.6;
      AN    I    100.1;
      AN    I      0.1;
      )     ;
      =     L      0.1;
      A     L      0.1;
      A     T    722;
      =     M   7002.6;
      A     L      0.1;
      BLD   102;
      L     S5T#0MS;
      SD    T    722;
      A     L      0.0;
      A(    ;
      O     DB327.DBX 1071.3;
      O     ;
      A     M   7002.7;
      AN    I    100.1;
      AN    I      0.1;
      )     ;
      =     L      0.1;
      A     L      0.1;
      A     T    723;
      =     M   7002.7;
      A     L      0.1;
      BLD   102;
      L     S5T#0MS;
      SD    T    723;
      A     L      0.0;
      A(    ;
      O     DB327.DBX 1073.3;
      O     ;
      A     M   7003.0;
      AN    I    100.1;
      AN    I      0.1;
      )     ;
      =     L      0.1;
      A     L      0.1;
      A     T    724;
      =     M   7003.0;
      A     L      0.1;
      BLD   102;
      L     S5T#0MS;
      SD    T    724;
      A     L      0.0;
      A(    ;
      O     DB327.DBX 1075.3;
      O     ;
      A     M   7003.1;
      AN    I    100.1;
      AN    I      0.1;
      )     ;
      =     L      0.1;
      A     L      0.1;
      A     T    725;
      =     M   7003.1;
      A     L      0.1;
      BLD   102;
      L     S5T#0MS;
      SD    T    725;
      A     L      0.0;
      A(    ;
      O     DB327.DBX 1077.3;
      O     ;
      A     M   7003.2;
      AN    I    100.1;
      AN    I      0.1;
      )     ;
      =     L      0.1;
      A     L      0.1;
      A     T    726;
      =     M   7003.2;
      A     L      0.1;
      BLD   102;
      L     S5T#0MS;
      SD    T    726;
      A     L      0.0;
      A(    ;
      O     DB327.DBX 1079.3;
      O     ;
      A     M   7003.3;
      AN    I    100.1;
      AN    I      0.1;
      )     ;
      =     L      0.1;
      A     L      0.1;
      A     T    727;
      AN    M      3.3;
      =     M   7003.3;
      A     L      0.1;
      BLD   102;
      L     S5T#0MS;
      SD    T    727;
      A     L      0.0;
      A(    ;
      O     DB327.DBX 1081.3;
      O     ;
      A     M   7003.4;
      AN    I    100.1;
      AN    I      0.1;
      )     ;
      =     L      0.1;
      A     L      0.1;
      A     T    728;
      AN    M      3.3;
      =     M   7003.4;
      A     L      0.1;
      BLD   102;
      L     S5T#0MS;
      SD    T    728;
      A     L      0.0;
      A(    ;
      O     DB327.DBX 1083.3;
      O     ;
      A     M   7003.5;
      AN    I    100.1;
      AN    I      0.1;
      )     ;
      =     L      0.1;
      A     L      0.1;
      A     T    729;
      AN    M      3.3;
      =     M   7003.5;
      A     L      0.1;
      BLD   102;
      L     S5T#0MS;
      SD    T    729;
NETWORK
TITLE =PROFINET ERROR(31~40)
//
//
      A     M      3.3;
      =     L      0.0;
      A     L      0.0;
      A(    ;
      O     DB327.DBX 1085.3;
      O     ;
      A     M   7003.6;
      AN    I    100.1;
      AN    I      0.1;
      )     ;
      =     L      0.1;
      A     L      0.1;
      A     T    730;
      AN    M      3.3;
      =     M   7003.6;
      A     L      0.1;
      BLD   102;
      L     S5T#0MS;
      SD    T    730;
      A     L      0.0;
      A(    ;
      O     DB327.DBX 1087.3;
      O     ;
      A     M   7003.7;
      AN    I    100.1;
      AN    I      0.1;
      )     ;
      =     L      0.1;
      A     L      0.1;
      A     T    731;
      AN    M      3.3;
      =     M   7003.7;
      A     L      0.1;
      BLD   102;
      L     S5T#0MS;
      SD    T    731;
      A     L      0.0;
      A(    ;
      O     DB327.DBX 1089.3;
      O     ;
      A     M   7004.0;
      AN    I    100.1;
      AN    I      0.1;
      )     ;
      =     L      0.1;
      A     L      0.1;
      A     T    732;
      AN    M      3.3;
      =     M   7004.0;
      A     L      0.1;
      BLD   102;
      L     S5T#0MS;
      SD    T    732;
      A     L      0.0;
      A(    ;
      O     DB327.DBX 1091.3;
      O     ;
      A     M   7004.1;
      AN    I    100.1;
      AN    I      0.1;
      )     ;
      =     L      0.1;
      A     L      0.1;
      A     T    733;
      AN    M      3.3;
      =     M   7004.1;
      A     L      0.1;
      BLD   102;
      L     S5T#0MS;
      SD    T    733;
      A     L      0.0;
      A(    ;
      O     DB327.DBX 1093.3;
      O     ;
      A     M   7004.2;
      AN    I    100.1;
      AN    I      0.1;
      )     ;
      =     L      0.1;
      A     L      0.1;
      A     T    734;
      AN    M      3.3;
      =     M   7004.2;
      A     L      0.1;
      BLD   102;
      L     S5T#0MS;
      SD    T    734;
      A     L      0.0;
      A(    ;
      O     DB327.DBX 1095.3;
      O     ;
      A     M   7004.3;
      AN    I    100.1;
      AN    I      0.1;
      )     ;
      =     L      0.1;
      A     L      0.1;
      A     T    735;
      AN    M      3.3;
      =     M   7004.3;
      A     L      0.1;
      BLD   102;
      L     S5T#0MS;
      SD    T    735;
      A     L      0.0;
      A(    ;
      O     DB327.DBX 1097.3;
      O     ;
      A     M   7004.4;
      AN    I    100.1;
      AN    I      0.1;
      )     ;
      =     L      0.1;
      A     L      0.1;
      A     T    736;
      AN    M      3.3;
      =     M   7004.4;
      A     L      0.1;
      BLD   102;
      L     S5T#0MS;
      SD    T    736;
      A     L      0.0;
      A(    ;
      O     DB327.DBX 1099.3;
      O     ;
      A     M   7004.5;
      AN    I    100.1;
      AN    I      0.1;
      )     ;
      =     L      0.1;
      A     L      0.1;
      A     T    737;
      AN    M      3.3;
      =     M   7004.5;
      A     L      0.1;
      BLD   102;
      L     S5T#0MS;
      SD    T    737;
      A     L      0.0;
      A(    ;
      O     DB327.DBX 1101.3;
      O     ;
      A     M   7004.6;
      AN    I    100.1;
      AN    I      0.1;
      )     ;
      =     L      0.1;
      A     L      0.1;
      A     T    738;
      AN    M      3.3;
      =     M   7004.6;
      A     L      0.1;
      BLD   102;
      L     S5T#0MS;
      SD    T    738;
      A     L      0.0;
      A(    ;
      O     DB327.DBX 1103.3;
      O     ;
      A     M   7004.7;
      AN    I    100.1;
      AN    I      0.1;
      )     ;
      =     L      0.1;
      A     L      0.1;
      A     T    739;
      AN    M      3.3;
      =     M   7004.7;
      A     L      0.1;
      BLD   102;
      L     S5T#0MS;
      SD    T    739;
NETWORK
TITLE =PROFINET ERROR(150~159)

      A     M      3.3;
      =     L      0.0;
      A     L      0.0;
      A(    ;
      O     DB327.DBX 1323.3;
      O     ;
      A     M   7018.5;
      AN    I    100.1;
      AN    I      0.1;
      )     ;
      =     L      0.1;
      A     L      0.1;
      A     T    849;
      AN    M      3.3;
      =     M   7018.5;
      A     L      0.1;
      BLD   102;
      L     S5T#0MS;
      SD    T    849;
      A     L      0.0;
      A(    ;
      O     DB327.DBX 1325.3;
      O     ;
      A     M   7018.6;
      AN    I    100.1;
      AN    I      0.1;
      )     ;
      =     L      0.1;
      A     L      0.1;
      A     T    850;
      AN    M      3.3;
      =     M   7018.6;
      A     L      0.1;
      BLD   102;
      L     S5T#0MS;
      SD    T    850;
      A     L      0.0;
      A(    ;
      O     DB327.DBX 1327.3;
      O     ;
      A     M   7018.7;
      AN    I    100.1;
      AN    I      0.1;
      )     ;
      =     L      0.1;
      A     L      0.1;
      A     T    851;
      AN    M      3.3;
      =     M   7018.7;
      A     L      0.1;
      BLD   102;
      L     S5T#0MS;
      SD    T    851;
      A     L      0.0;
      A(    ;
      O     DB327.DBX 1329.3;
      O     ;
      A     M   7019.0;
      AN    I    100.1;
      AN    I      0.1;
      )     ;
      =     L      0.1;
      A     L      0.1;
      A     T    852;
      AN    M      3.3;
      =     M   7019.0;
      A     L      0.1;
      BLD   102;
      L     S5T#0MS;
      SD    T    852;
      A     L      0.0;
      A(    ;
      O     DB327.DBX 1331.3;
      O     ;
      A     M   7019.1;
      AN    I    100.1;
      AN    I      0.1;
      )     ;
      =     L      0.1;
      A     L      0.1;
      A     T    853;
      AN    M      3.3;
      =     M   7019.1;
      A     L      0.1;
      BLD   102;
      L     S5T#0MS;
      SD    T    853;
      A     L      0.0;
      A(    ;
      O     DB327.DBX 1333.3;
      O     ;
      A     M   7019.2;
      AN    I    100.1;
      AN    I      0.1;
      )     ;
      =     L      0.1;
      A     L      0.1;
      A     T    854;
      AN    M      3.3;
      =     M   7019.2;
      A     L      0.1;
      BLD   102;
      L     S5T#0MS;
      SD    T    854;
      A     L      0.0;
      A(    ;
      O     DB327.DBX 1335.3;
      O     ;
      A     M   7019.3;
      AN    I    100.1;
      AN    I      0.1;
      )     ;
      =     L      0.1;
      A     L      0.1;
      A     T    855;
      AN    M      3.3;
      =     M   7019.3;
      A     L      0.1;
      BLD   102;
      L     S5T#0MS;
      SD    T    855;
      A     L      0.0;
      A(    ;
      O     DB327.DBX 1337.3;
      O     ;
      A     M   7019.4;
      AN    I    100.1;
      AN    I      0.1;
      )     ;
      =     L      0.1;
      A     L      0.1;
      A     T    856;
      AN    M      3.3;
      =     M   7019.4;
      A     L      0.1;
      BLD   102;
      L     S5T#0MS;
      SD    T    856;
      A     L      0.0;
      A(    ;
      O     DB327.DBX 1339.3;
      O     ;
      A     M   7019.5;
      AN    I    100.1;
      AN    I      0.1;
      )     ;
      =     L      0.1;
      A     L      0.1;
      A     T    857;
      AN    M      3.3;
      =     M   7019.5;
      A     L      0.1;
      BLD   102;
      L     S5T#0MS;
      SD    T    857;
      A     L      0.0;
      A(    ;
      O     DB327.DBX 1341.3;
      O     ;
      A     M   7019.6;
      AN    I    100.1;
      AN    I      0.1;
      )     ;
      =     L      0.1;
      A     L      0.1;
      A     T    858;
      AN    M      3.3;
      =     M   7019.6;
      A     L      0.1;
      BLD   102;
      L     S5T#0MS;
      SD    T    858;
NETWORK
TITLE =CP TRIP(20~29)
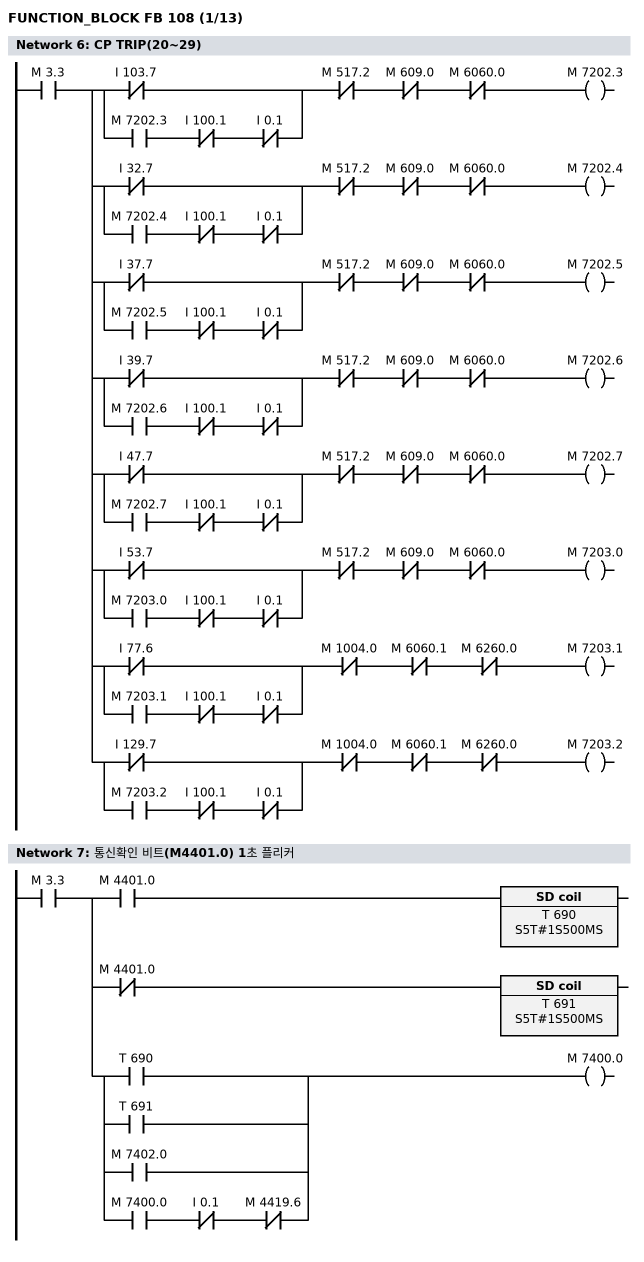

      A     M      3.3;
      =     L      0.0;
      A     L      0.0;
      A(    ;
      ON    I    103.7;
      O     ;
      A     M   7202.3;
      AN    I    100.1;
      AN    I      0.1;
      )     ;
      AN    M    517.2;
      AN    M    609.0;
      AN    M   6060.0;
      =     M   7202.3;
      A     L      0.0;
      A(    ;
      ON    I     32.7;
      O     ;
      A     M   7202.4;
      AN    I    100.1;
      AN    I      0.1;
      )     ;
      AN    M    517.2;
      AN    M    609.0;
      AN    M   6060.0;
      =     M   7202.4;
      A     L      0.0;
      A(    ;
      ON    I     37.7;
      O     ;
      A     M   7202.5;
      AN    I    100.1;
      AN    I      0.1;
      )     ;
      AN    M    517.2;
      AN    M    609.0;
      AN    M   6060.0;
      =     M   7202.5;
      A     L      0.0;
      A(    ;
      ON    I     39.7;
      O     ;
      A     M   7202.6;
      AN    I    100.1;
      AN    I      0.1;
      )     ;
      AN    M    517.2;
      AN    M    609.0;
      AN    M   6060.0;
      =     M   7202.6;
      A     L      0.0;
      A(    ;
      ON    I     47.7;
      O     ;
      A     M   7202.7;
      AN    I    100.1;
      AN    I      0.1;
      )     ;
      AN    M    517.2;
      AN    M    609.0;
      AN    M   6060.0;
      =     M   7202.7;
      A     L      0.0;
      A(    ;
      ON    I     53.7;
      O     ;
      A     M   7203.0;
      AN    I    100.1;
      AN    I      0.1;
      )     ;
      AN    M    517.2;
      AN    M    609.0;
      AN    M   6060.0;
      =     M   7203.0;
      A     L      0.0;
      A(    ;
      ON    I     77.6;
      O     ;
      A     M   7203.1;
      AN    I    100.1;
      AN    I      0.1;
      )     ;
      AN    M   1004.0;
      AN    M   6060.1;
      AN    M   6260.0;
      =     M   7203.1;
      A     L      0.0;
      A(    ;
      ON    I    129.7;
      O     ;
      A     M   7203.2;
      AN    I    100.1;
      AN    I      0.1;
      )     ;
      AN    M   1004.0;
      AN    M   6060.1;
      AN    M   6260.0;
      =     M   7203.2;
NETWORK
TITLE =통신확인 비트(M4401.0) 1초 플리커
//
//
      A     M      3.3;
      =     L      0.0;
      A     L      0.0;
      A     M   4401.0;
      L     S5T#1S500MS;
      SD    T    690;
      A     L      0.0;
      AN    M   4401.0;
      L     S5T#1S500MS;
      SD    T    691;
      A     L      0.0;
      A(    ;
      O     T    690;
      O     T    691;
      O     M   7402.0;
      O     ;
      A     M   7400.0;
      AN    I      0.1;
      AN    M   4419.6;
      )     ;
      =     M   7400.0;
NETWORK
TITLE =통신확인 비트(M4701.0) 1초 플리커
//
//
//
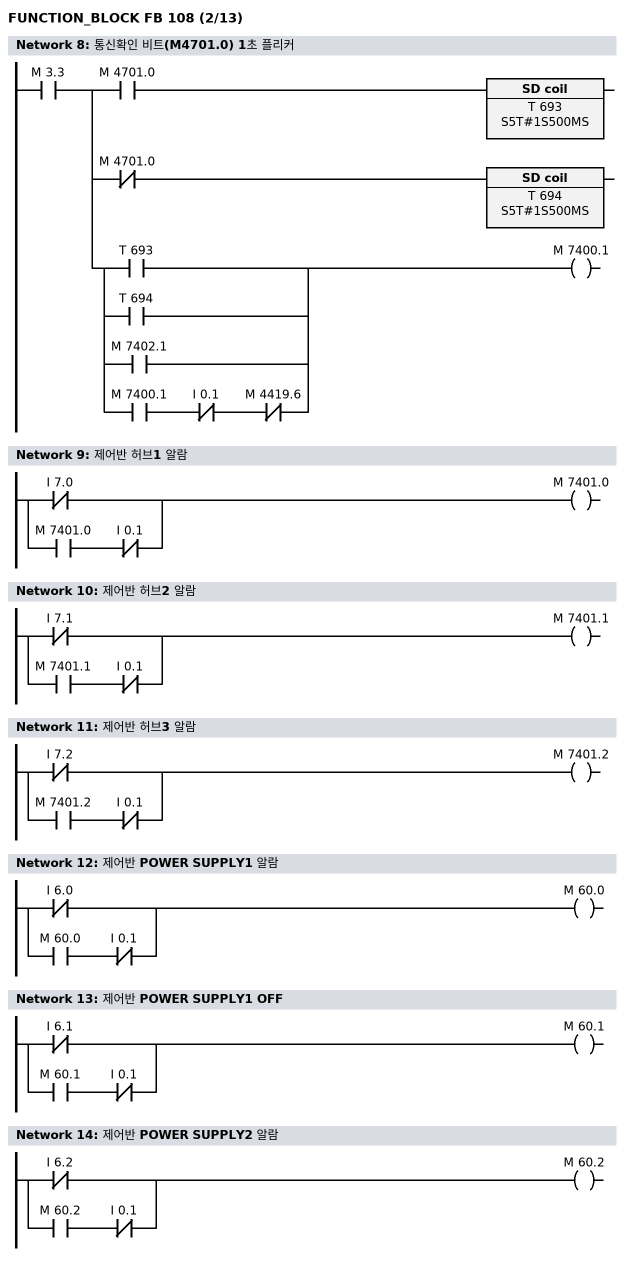
      A     M      3.3;
      =     L      0.0;
      A     L      0.0;
      A     M   4701.0;
      L     S5T#1S500MS;
      SD    T    693;
      A     L      0.0;
      AN    M   4701.0;
      L     S5T#1S500MS;
      SD    T    694;
      A     L      0.0;
      A(    ;
      O     T    693;
      O     T    694;
      O     M   7402.1;
      O     ;
      A     M   7400.1;
      AN    I      0.1;
      AN    M   4419.6;
      )     ;
      =     M   7400.1;
NETWORK
TITLE =제어반 허브1 알람

      ON    I      7.0;
      O     ;
      A     M   7401.0;
      AN    I      0.1;
      =     M   7401.0;
NETWORK
TITLE =제어반 허브2 알람

      ON    I      7.1;
      O     ;
      A     M   7401.1;
      AN    I      0.1;
      =     M   7401.1;
NETWORK
TITLE =제어반 허브3 알람

      ON    I      7.2;
      O     ;
      A     M   7401.2;
      AN    I      0.1;
      =     M   7401.2;
NETWORK
TITLE =제어반 POWER SUPPLY1 알람

      ON    I      6.0;
      O     ;
      A     M     60.0;
      AN    I      0.1;
      =     M     60.0;
NETWORK
TITLE =제어반 POWER SUPPLY1 OFF

      ON    I      6.1;
      O     ;
      A     M     60.1;
      AN    I      0.1;
      =     M     60.1;
NETWORK
TITLE =제어반 POWER SUPPLY2 알람
//
//
      ON    I      6.2;
      O     ;
      A     M     60.2;
      AN    I      0.1;
      =     M     60.2;
NETWORK
TITLE =제어반 POWER SUPPLY2 OFF
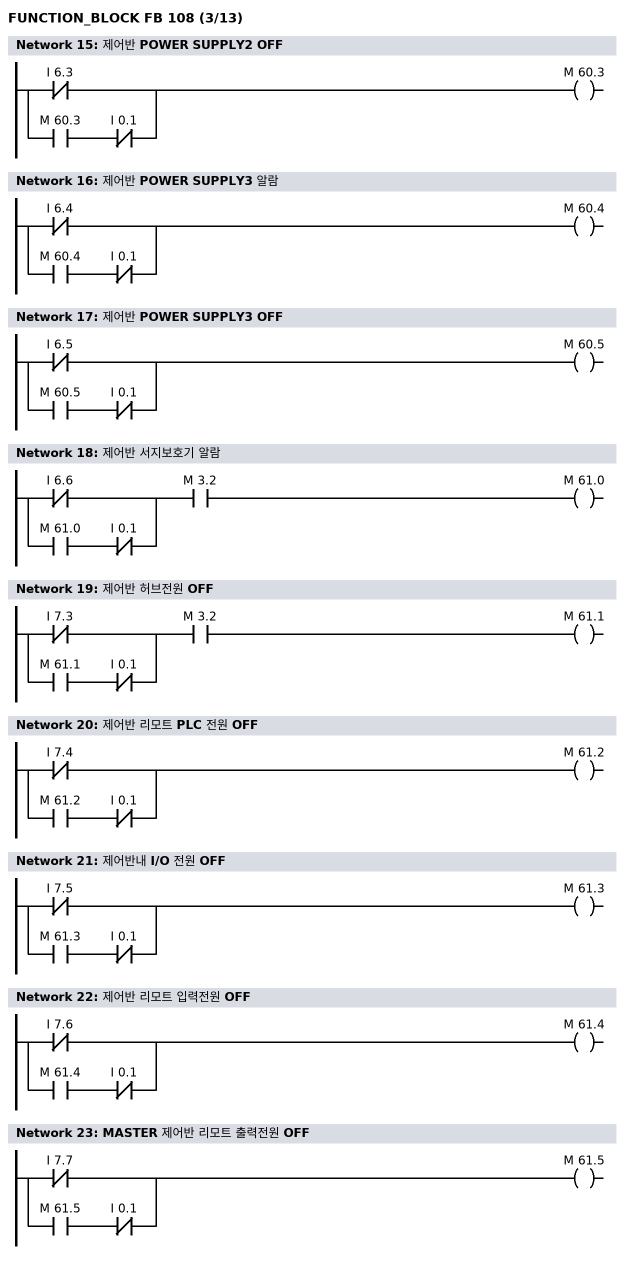

      ON    I      6.3;
      O     ;
      A     M     60.3;
      AN    I      0.1;
      =     M     60.3;
NETWORK
TITLE =제어반 POWER SUPPLY3 알람
//
//
      ON    I      6.4;
      O     ;
      A     M     60.4;
      AN    I      0.1;
      =     M     60.4;
NETWORK
TITLE =제어반 POWER SUPPLY3 OFF

      ON    I      6.5;
      O     ;
      A     M     60.5;
      AN    I      0.1;
      =     M     60.5;
NETWORK
TITLE =제어반 서지보호기 알람

      A(    ;
      ON    I      6.6;
      O     ;
      A     M     61.0;
      AN    I      0.1;
      )     ;
      A     M      3.2;
      =     M     61.0;
NETWORK
TITLE =제어반 허브전원 OFF

      A(    ;
      ON    I      7.3;
      O     ;
      A     M     61.1;
      AN    I      0.1;
      )     ;
      A     M      3.2;
      =     M     61.1;
NETWORK
TITLE =제어반 리모트 PLC 전원 OFF

      ON    I      7.4;
      O     ;
      A     M     61.2;
      AN    I      0.1;
      =     M     61.2;
NETWORK
TITLE =제어반내 I/O 전원 OFF

      ON    I      7.5;
      O     ;
      A     M     61.3;
      AN    I      0.1;
      =     M     61.3;
NETWORK
TITLE =제어반 리모트 입력전원 OFF

      ON    I      7.6;
      O     ;
      A     M     61.4;
      AN    I      0.1;
      =     M     61.4;
NETWORK
TITLE =MASTER 제어반 리모트 출력전원 OFF

